  MoveL 658 to (4.03, 195.62, 30) mm, rotated rx 180 ry 50 rz -176.42 deg; joints [-18.981, -46.82, 111.254, 128.122, 73.547, 109.847, -1353.581]
  MoveL 659 to (9.5, 196.25, 40) mm, rotated rx 180 ry 50 rz -171.53 deg; joints [-18.576, -46.815, 111.235, 128.515, 73.401, 109.745, -1358.473]
  MoveL 660 to (15.19, 197.47, 50) mm, rotated rx -180 ry 50 rz -166.35 deg; joints [-18.172, -46.809, 111.211, 128.908, 73.253, 109.646, -1363.653]
  MoveL 661 to (21, 199.35, 60) mm, rotated rx -180 ry 50 rz -160.91 deg; joints [-17.768, -46.804, 111.18, 129.3, 73.102, 109.552, -1369.094]
  MoveL 662 to (26.8, 201.92, 70) mm, rotated rx 180 ry 50 rz -155.23 deg; joints [-17.364, -46.8, 111.144, 129.691, 72.947, 109.461, -1374.769]
  MoveL 663 to (32.46, 205.23, 80) mm, rotated rx -180 ry 50 rz -149.35 deg; joints [-16.96, -46.796, 111.102, 130.08, 72.788, 109.375, -1380.653]
  MoveL 664 to (37.86, 209.24, 90) mm, rotated rx 180 ry 50 rz -143.28 deg; joints [-16.557, -46.793, 111.054, 130.468, 72.625, 109.292, -1386.718]
  MoveL 665 to (42.85, 213.95, 100) mm, rotated rx 180 ry 50 rz -137.06 deg; joints [-16.154, -46.79, 110.999, 130.854, 72.459, 109.214, -1392.941]
  MoveL 666 to (47.33, 219.29, 110) mm, rotated rx -180 ry 50 rz -130.7 deg; joints [-15.751, -46.788, 110.939, 131.239, 72.288, 109.139, -1399.296]
  MoveL 667 to (51.17, 225.17, 120) mm, rotated rx -180 ry 50 rz -124.24 deg; joints [-15.349, -46.786, 110.873, 131.623, 72.114, 109.067, -1405.756]
  MoveL 668 to (54.3, 231.49, 130) mm, rotated rx -180 ry 50 rz -117.7 deg; joints [-14.948, -46.784, 110.801, 132.005, 71.937, 108.999, -1412.295]
  MoveL 669 to (56.65, 238.12, 140) mm, rotated rx 180 ry 50 rz -111.11 deg; joints [-14.546, -46.781, 110.723, 132.386, 71.756, 108.933, -1418.886]
  MoveL 670 to (58.18, 244.95, 150) mm, rotated rx 180 ry 50 rz -104.5 deg; joints [-14.146, -46.776, 110.639, 132.766, 71.573, 108.868, -1425.497]
  MoveL 671 to (58.89, 251.83, 160) mm, rotated rx 180 ry 50 rz -97.9 deg; joints [-13.746, -46.768, 110.548, 133.145, 71.387, 108.806, -1432.098]
  MoveL 672 to (58.8, 258.62, 170) mm, rotated rx -180 ry 50 rz -91.34 deg; joints [-13.346, -46.758, 110.451, 133.523, 71.199, 108.744, -1438.655]
  MoveL 673 to (57.96, 265.2, 180) mm, rotated rx 180 ry 50 rz -84.87 deg; joints [-12.947, -46.744, 110.348, 133.901, 71.009, 108.683, -1445.13]
  MoveL 674 to (56.44, 271.47, 190) mm, rotated rx 180 ry 50 rz -78.51 deg; joints [-12.549, -46.726, 110.239, 134.277, 70.818, 108.622, -1451.486]
  MoveL 675 to (54.33, 277.32, 200) mm, rotated rx -180 ry 50 rz -72.32 deg; joints [-12.152, -46.703, 110.123, 134.653, 70.627, 108.56, -1457.679]
  MoveL 676 to (51.74, 282.68, 210) mm, rotated rx 180 ry 50 rz -66.33 deg; joints [-11.755, -46.675, 110.001, 135.028, 70.435, 108.498, -1463.668]
  MoveL 677 to (48.8, 287.5, 220) mm, rotated rx -180 ry 50 rz -60.59 deg; joints [-11.359, -46.641, 109.872, 135.403, 70.242, 108.434, -1469.406]
  MoveL 678 to (45.62, 291.76, 230) mm, rotated rx 180 ry 50 rz -55.15 deg; joints [-10.964, -46.601, 109.737, 135.778, 70.049, 108.37, -1474.846]
  MoveL 679 to (42.34, 295.45, 240) mm, rotated rx 180 ry 50 rz -50.06 deg; joints [-10.57, -46.555, 109.596, 136.152, 69.856, 108.304, -1479.941]
  MoveL 680 to (39.07, 298.58, 250) mm, rotated rx 180 ry 50 rz -45.36 deg; joints [-10.177, -46.504, 109.448, 136.525, 69.663, 108.237, -1484.643]
  MoveL 681 to (35.92, 301.18, 260) mm, rotated rx -180 ry 50 rz -41.09 deg; joints [-9.784, -46.446, 109.294, 136.898, 69.47, 108.169, -1488.905]
  MoveL 682 to (33, 303.28, 270) mm, rotated rx 180 ry 50 rz -37.32 deg; joints [-9.393, -46.383, 109.133, 137.271, 69.277, 108.1, -1492.679]
  MoveL 683 to (30.4, 304.94, 280) mm, rotated rx 180 ry 50 rz -34.08 deg; joints [-9.003, -46.315, 108.966, 137.642, 69.083, 108.031, -1495.919]
  MoveL 684 to (28.22, 306.19, 290) mm, rotated rx 180 ry 50 rz -31.42 deg; joints [-8.613, -46.241, 108.793, 138.013, 68.889, 107.96, -1498.582]
  MoveL 685 to (-21.11, 309.47, 290) mm, rotated rx -180 ry 50 rz 23.11 deg; joints [-8.613, -46.26, 108.794, 138.009, 68.876, 107.972, -1553.11]
  Set speed (60.0 mm/s)
  MoveL 686 to (-18.74, 310.33, 280) mm, rotated rx -180 ry 50 rz 20.42 deg; joints [-9.003, -46.345, 108.968, 137.635, 69.063, 108.051, -1550.424]
  MoveL 687 to (-15.8, 311.23, 270) mm, rotated rx -180 ry 50 rz 17.14 deg; joints [-9.393, -46.428, 109.136, 137.26, 69.247, 108.13, -1547.138]
  MoveL 688 to (-12.3, 312.09, 260) mm, rotated rx 180 ry 50 rz 13.29 deg; joints [-9.784, -46.507, 109.298, 136.884, 69.429, 108.211, -1543.29]
  MoveL 689 to (-8.28, 312.8, 250) mm, rotated rx -180 ry 50 rz 8.92 deg; joints [-10.177, -46.583, 109.454, 136.506, 69.61, 108.292, -1538.917]
  MoveL 690 to (-3.78, 313.26, 240) mm, rotated rx -180 ry 50 rz 4.06 deg; joints [-10.57, -46.655, 109.603, 136.128, 69.79, 108.372, -1534.059]
  MoveL 691 to (1.16, 313.37, 230) mm, rotated rx 180 ry 50 rz -1.24 deg; joints [-10.964, -46.722, 109.746, 135.749, 69.969, 108.453, -1528.756]
  MoveL 692 to (6.46, 313.03, 220) mm, rotated rx 180 ry 50 rz -6.95 deg; joints [-11.359, -46.783, 109.883, 135.37, 70.148, 108.533, -1523.053]
  MoveL 693 to (12.04, 312.14, 210) mm, rotated rx 180 ry 50 rz -13.01 deg; joints [-11.755, -46.838, 110.013, 134.99, 70.327, 108.612, -1516.995]
  MoveL 694 to (17.8, 310.63, 200) mm, rotated rx 180 ry 50 rz -19.37 deg; joints [-12.152, -46.887, 110.136, 134.61, 70.507, 108.689, -1510.629]
  MoveL 695 to (23.62, 308.44, 190) mm, rotated rx -180 ry 50 rz -25.99 deg; joints [-12.549, -46.929, 110.254, 134.23, 70.687, 108.765, -1504.006]
  MoveL 696 to (29.38, 305.54, 180) mm, rotated rx -180 ry 50 rz -32.82 deg; joints [-12.947, -46.964, 110.364, 133.85, 70.868, 108.838, -1497.176]
  MoveL 697 to (34.94, 301.92, 170) mm, rotated rx -180 ry 50 rz -39.81 deg; joints [-13.346, -46.992, 110.469, 133.47, 71.049, 108.911, -1490.188]
  MoveL 698 to (40.17, 297.58, 160) mm, rotated rx 180 ry 50 rz -46.91 deg; joints [-13.746, -47.014, 110.566, 133.089, 71.231, 108.981, -1483.094]
  MoveL 699 to (44.94, 292.58, 150) mm, rotated rx -180 ry 50 rz -54.06 deg; joints [-14.146, -47.029, 110.658, 132.709, 71.413, 109.05, -1475.941]
  MoveL 700 to (49.15, 286.99, 140) mm, rotated rx -180 ry 50 rz -61.23 deg; joints [-14.546, -47.038, 110.743, 132.328, 71.596, 109.118, -1468.774]
  MoveL 701 to (52.68, 280.9, 130) mm, rotated rx -180 ry 50 rz -68.36 deg; joints [-14.948, -47.042, 110.821, 131.947, 71.777, 109.185, -1461.638]
  MoveL 702 to (55.46, 274.42, 120) mm, rotated rx -180 ry 50 rz -75.43 deg; joints [-15.349, -47.042, 110.893, 131.566, 71.958, 109.252, -1454.572]
  MoveL 703 to (57.44, 267.68, 110) mm, rotated rx 180 ry 50 rz -82.39 deg; joints [-15.751, -47.037, 110.959, 131.184, 72.137, 109.32, -1447.613]
  MoveL 704 to (58.6, 260.81, 100) mm, rotated rx 180 ry 50 rz -89.21 deg; joints [-16.154, -47.029, 111.018, 130.801, 72.315, 109.388, -1440.794]
  MoveL 705 to (58.95, 253.96, 90) mm, rotated rx -180 ry 50 rz -95.85 deg; joints [-16.557, -47.019, 111.072, 130.418, 72.49, 109.458, -1434.147]
  MoveL 706 to (58.51, 247.24, 80) mm, rotated rx -180 ry 50 rz -102.3 deg; joints [-16.96, -47.007, 111.119, 130.034, 72.663, 109.53, -1427.701]
  MoveL 707 to (57.35, 240.79, 70) mm, rotated rx 180 ry 50 rz -108.52 deg; joints [-17.364, -46.993, 111.16, 129.648, 72.833, 109.604, -1421.482]
  MoveL 708 to (55.55, 234.7, 60) mm, rotated rx -180 ry 50 rz -114.48 deg; joints [-17.768, -46.979, 111.195, 129.262, 73, 109.682, -1415.517]
  MoveL 709 to (53.21, 229.07, 50) mm, rotated rx 180 ry 50 rz -120.17 deg; joints [-18.172, -46.965, 111.224, 128.875, 73.164, 109.762, -1409.83]
  MoveL 710 to (50.45, 223.94, 40) mm, rotated rx 180 ry 50 rz -125.55 deg; joints [-18.576, -46.951, 111.246, 128.486, 73.324, 109.847, -1404.447]
  MoveL 711 to (47.39, 219.37, 30) mm, rotated rx 180 ry 50 rz -130.61 deg; joints [-18.981, -46.936, 111.263, 128.097, 73.481, 109.934, -1399.391]
  MoveL 712 to (44.15, 215.37, 20) mm, rotated rx 180 ry 50 rz -135.31 deg; joints [-19.385, -46.922, 111.274, 127.706, 73.634, 110.026, -1394.688]
  MoveL 713 to (40.85, 211.93, 10) mm, rotated rx 180 ry 50 rz -139.64 deg; joints [-19.79, -46.908, 111.279, 127.315, 73.785, 110.121, -1390.363]
  MoveL 714 to (37.62, 209.05, 0) mm, rotated rx 180 ry 50 rz -143.56 deg; joints [-20.194, -46.894, 111.278, 126.922, 73.932, 110.22, -1386.442]
  MoveL 715 to (-21.11, 309.47, 290) mm, rotated rx -180 ry 50 rz 23.11 deg; joints [-8.613, -46.26, 108.794, 138.009, 68.876, 107.972, -1553.11]
  Set speed (60.0 mm/s)
  MoveL 716 to (-34.79, 325.15, 290) mm, rotated rx 180 ry 50 rz 28.1 deg; joints [-8.613, -45.167, 108.701, 138.262, 69.621, 107.259, -1558.101]
  MoveL 717 to (37.62, 209.05, 0) mm, rotated rx 180 ry 50 rz -143.56 deg; joints [-20.194, -46.894, 111.278, 126.922, 73.932, 110.22, -1386.442]
  Set speed (60.0 mm/s)
  MoveL 718 to (55.59, 198.58, 0) mm, rotated rx 180 ry 50 rz -137.85 deg; joints [-20.194, -45.798, 111.172, 127.145, 74.528, 109.399, -1392.15]
  MoveL 719 to (37.62, 209.05, 0) mm, rotated rx 180 ry 50 rz -143.56 deg; joints [-20.194, -46.894, 111.278, 126.922, 73.932, 110.22, -1386.442]
  Set speed (60.0 mm/s)
  MoveL 720 to (40.85, 211.93, 10) mm, rotated rx 180 ry 50 rz -139.64 deg; joints [-19.79, -46.908, 111.279, 127.315, 73.785, 110.121, -1390.363]
  MoveL 721 to (44.15, 215.37, 20) mm, rotated rx 180 ry 50 rz -135.31 deg; joints [-19.385, -46.922, 111.274, 127.706, 73.634, 110.026, -1394.688]
  MoveL 722 to (47.39, 219.37, 30) mm, rotated rx 180 ry 50 rz -130.61 deg; joints [-18.981, -46.936, 111.263, 128.097, 73.481, 109.934, -1399.391]
  MoveL 723 to (50.45, 223.94, 40) mm, rotated rx 180 ry 50 rz -125.55 deg; joints [-18.576, -46.951, 111.246, 128.486, 73.324, 109.847, -1404.447]
  MoveL 724 to (53.21, 229.07, 50) mm, rotated rx 180 ry 50 rz -120.17 deg; joints [-18.172, -46.965, 111.224, 128.875, 73.164, 109.762, -1409.83]
  MoveL 725 to (55.55, 234.7, 60) mm, rotated rx -180 ry 50 rz -114.48 deg; joints [-17.768, -46.979, 111.195, 129.262, 73, 109.682, -1415.517]
  MoveL 726 to (57.35, 240.79, 70) mm, rotated rx -180 ry 50 rz -108.52 deg; joints [-17.364, -46.993, 111.16, 129.648, 72.833, 109.604, -1421.482]
  MoveL 727 to (58.51, 247.24, 80) mm, rotated rx 180 ry 50 rz -102.3 deg; joints [-16.96, -47.007, 111.119, 130.034, 72.663, 109.53, -1427.701]
  MoveL 728 to (58.95, 253.96, 90) mm, rotated rx 180 ry 50 rz -95.85 deg; joints [-16.557, -47.019, 111.072, 130.418, 72.49, 109.458, -1434.147]
  MoveL 729 to (58.6, 260.81, 100) mm, rotated rx 180 ry 50 rz -89.21 deg; joints [-16.154, -47.029, 111.018, 130.801, 72.315, 109.388, -1440.794]
  MoveL 730 to (57.44, 267.68, 110) mm, rotated rx 180 ry 50 rz -82.39 deg; joints [-15.751, -47.037, 110.959, 131.184, 72.137, 109.32, -1447.613]
  MoveL 731 to (55.46, 274.42, 120) mm, rotated rx 180 ry 50 rz -75.43 deg; joints [-15.349, -47.042, 110.893, 131.566, 71.958, 109.252, -1454.572]
  MoveL 732 to (52.68, 280.9, 130) mm, rotated rx -180 ry 50 rz -68.36 deg; joints [-14.948, -47.042, 110.821, 131.947, 71.777, 109.185, -1461.638]
  MoveL 733 to (49.15, 286.99, 140) mm, rotated rx -180 ry 50 rz -61.23 deg; joints [-14.546, -47.038, 110.743, 132.328, 71.596, 109.118, -1468.774]
  MoveL 734 to (44.94, 292.58, 150) mm, rotated rx -180 ry 50 rz -54.06 deg; joints [-14.146, -47.029, 110.658, 132.709, 71.413, 109.05, -1475.941]
  MoveL 735 to (40.17, 297.58, 160) mm, rotated rx -180 ry 50 rz -46.91 deg; joints [-13.746, -47.014, 110.566, 133.089, 71.231, 108.981, -1483.094]
  MoveL 736 to (34.94, 301.92, 170) mm, rotated rx 180 ry 50 rz -39.81 deg; joints [-13.346, -46.992, 110.469, 133.47, 71.049, 108.911, -1490.188]
  MoveL 737 to (29.38, 305.54, 180) mm, rotated rx 180 ry 50 rz -32.82 deg; joints [-12.947, -46.964, 110.364, 133.85, 70.868, 108.838, -1497.176]
  MoveL 738 to (23.62, 308.44, 190) mm, rotated rx 180 ry 50 rz -25.99 deg; joints [-12.549, -46.929, 110.254, 134.23, 70.687, 108.765, -1504.006]
  MoveL 739 to (17.8, 310.63, 200) mm, rotated rx -180 ry 50 rz -19.37 deg; joints [-12.152, -46.887, 110.136, 134.61, 70.507, 108.689, -1510.629]
  MoveL 740 to (12.04, 312.14, 210) mm, rotated rx 180 ry 50 rz -13.01 deg; joints [-11.755, -46.838, 110.013, 134.99, 70.327, 108.612, -1516.995]
  MoveL 741 to (6.46, 313.03, 220) mm, rotated rx 180 ry 50 rz -6.95 deg; joints [-11.359, -46.783, 109.883, 135.37, 70.148, 108.533, -1523.053]
  MoveL 742 to (1.16, 313.37, 230) mm, rotated rx 180 ry 50 rz -1.24 deg; joints [-10.964, -46.722, 109.746, 135.749, 69.969, 108.453, -1528.756]
  MoveL 743 to (-3.78, 313.26, 240) mm, rotated rx 180 ry 50 rz 4.06 deg; joints [-10.57, -46.655, 109.603, 136.128, 69.79, 108.372, -1534.059]
  MoveL 744 to (-8.28, 312.8, 250) mm, rotated rx 180 ry 50 rz 8.92 deg; joints [-10.177, -46.583, 109.454, 136.506, 69.61, 108.292, -1538.917]
  MoveL 745 to (-12.3, 312.09, 260) mm, rotated rx -180 ry 50 rz 13.29 deg; joints [-9.784, -46.507, 109.298, 136.884, 69.429, 108.211, -1543.29]
  MoveL 746 to (-15.8, 311.23, 270) mm, rotated rx -180 ry 50 rz 17.14 deg; joints [-9.393, -46.428, 109.136, 137.26, 69.247, 108.13, -1547.138]
  MoveL 747 to (-18.74, 310.33, 280) mm, rotated rx -180 ry 50 rz 20.42 deg; joints [-9.003, -46.345, 108.968, 137.635, 69.063, 108.051, -1550.424]
  MoveL 748 to (-21.11, 309.47, 290) mm, rotated rx -180 ry 50 rz 23.11 deg; joints [-8.613, -46.26, 108.794, 138.009, 68.876, 107.972, -1553.11]
  MoveL 749 to (-34.79, 325.15, 290) mm, rotated rx 180 ry 50 rz 28.1 deg; joints [-8.613, -45.167, 108.701, 138.262, 69.621, 107.259, -1558.101]
  Set speed (60.0 mm/s)
  MoveL 750 to (-31.73, 326.57, 280) mm, rotated rx 180 ry 50 rz 25.49 deg; joints [-9.003, -45.252, 108.876, 137.888, 69.803, 107.332, -1555.486]
  MoveL 751 to (-27.92, 328.13, 270) mm, rotated rx -180 ry 50 rz 22.29 deg; joints [-9.393, -45.334, 109.044, 137.512, 69.984, 107.407, -1552.288]
  MoveL 752 to (-23.38, 329.69, 260) mm, rotated rx 180 ry 50 rz 18.54 deg; joints [-9.784, -45.413, 109.206, 137.135, 70.162, 107.483, -1548.542]
  MoveL 753 to (-18.11, 331.13, 250) mm, rotated rx 180 ry 50 rz 14.29 deg; joints [-10.177, -45.49, 109.362, 136.757, 70.338, 107.56, -1544.286]
  MoveL 754 to (-12.17, 332.29, 240) mm, rotated rx -180 ry 50 rz 9.56 deg; joints [-10.57, -45.562, 109.511, 136.378, 70.513, 107.636, -1539.557]
  MoveL 755 to (-5.61, 333.04, 230) mm, rotated rx -180 ry 50 rz 4.39 deg; joints [-10.964, -45.629, 109.655, 135.998, 70.687, 107.713, -1534.392]
  MoveL 756 to (1.49, 333.22, 220) mm, rotated rx 180 ry 50 rz -1.17 deg; joints [-11.359, -45.692, 109.791, 135.618, 70.861, 107.79, -1528.834]
  MoveL 757 to (9.03, 332.72, 210) mm, rotated rx 180 ry 50 rz -7.08 deg; joints [-11.755, -45.749, 109.922, 135.237, 71.034, 107.865, -1522.922]
  MoveL 758 to (16.88, 331.41, 200) mm, rotated rx -180 ry 50 rz -13.3 deg; joints [-12.152, -45.799, 110.045, 134.856, 71.208, 107.94, -1516.702]
  MoveL 759 to (24.89, 329.2, 190) mm, rotated rx -180 ry 50 rz -19.78 deg; joints [-12.549, -45.843, 110.162, 134.474, 71.382, 108.013, -1510.217]
  MoveL 760 to (32.91, 326.04, 180) mm, rotated rx 180 ry 50 rz -26.49 deg; joints [-12.947, -45.88, 110.273, 134.093, 71.557, 108.084, -1503.513]
  MoveL 761 to (40.75, 321.89, 170) mm, rotated rx 180 ry 50 rz -33.36 deg; joints [-13.346, -45.91, 110.377, 133.711, 71.732, 108.154, -1496.637]
  MoveL 762 to (48.24, 316.75, 160) mm, rotated rx -180 ry 50 rz -40.37 deg; joints [-13.746, -45.934, 110.474, 133.329, 71.908, 108.222, -1489.635]
  MoveL 763 to (55.2, 310.67, 150) mm, rotated rx -180 ry 50 rz -47.45 deg; joints [-14.146, -45.95, 110.565, 132.947, 72.084, 108.289, -1482.551]
  MoveL 764 to (61.48, 303.74, 140) mm, rotated rx -180 ry 50 rz -54.57 deg; joints [-14.546, -45.961, 110.649, 132.565, 72.26, 108.354, -1475.431]
  MoveL 765 to (66.92, 296.06, 130) mm, rotated rx -180 ry 50 rz -61.68 deg; joints [-14.948, -45.965, 110.727, 132.183, 72.436, 108.419, -1468.317]
  MoveL 766 to (71.41, 287.77, 120) mm, rotated rx 180 ry 50 rz -68.75 deg; joints [-15.349, -45.965, 110.798, 131.8, 72.611, 108.483, -1461.249]
  MoveL 767 to (74.87, 279.04, 110) mm, rotated rx -180 ry 50 rz -75.73 deg; joints [-15.751, -45.96, 110.863, 131.417, 72.785, 108.547, -1454.266]
  MoveL 768 to (77.24, 270.04, 100) mm, rotated rx 180 ry 50 rz -82.6 deg; joints [-16.154, -45.952, 110.921, 131.033, 72.957, 108.612, -1447.404]
  MoveL 769 to (78.53, 260.95, 90) mm, rotated rx -180 ry 50 rz -89.3 deg; joints [-16.557, -45.941, 110.974, 130.648, 73.127, 108.678, -1440.696]
  MoveL 770 to (78.77, 251.96, 80) mm, rotated rx 180 ry 50 rz -95.83 deg; joints [-16.96, -45.927, 111.02, 130.263, 73.295, 108.746, -1434.174]
  MoveL 771 to (78, 243.23, 70) mm, rotated rx -180 ry 50 rz -102.13 deg; joints [-17.364, -45.912, 111.06, 129.877, 73.461, 108.816, -1427.868]
  MoveL 772 to (76.35, 234.91, 60) mm, rotated rx -180 ry 50 rz -108.19 deg; joints [-17.768, -45.896, 111.093, 129.49, 73.623, 108.889, -1421.808]
  MoveL 773 to (73.92, 227.12, 50) mm, rotated rx 180 ry 50 rz -113.98 deg; joints [-18.172, -45.88, 111.121, 129.101, 73.782, 108.965, -1416.021]
  MoveL 774 to (70.87, 219.96, 40) mm, rotated rx -180 ry 50 rz -119.46 deg; joints [-18.576, -45.863, 111.143, 128.712, 73.938, 109.045, -1410.535]
  MoveL 775 to (67.34, 213.5, 30) mm, rotated rx 180 ry 50 rz -124.62 deg; joints [-18.981, -45.847, 111.159, 128.322, 74.09, 109.128, -1405.378]
  MoveL 776 to (63.51, 207.78, 20) mm, rotated rx 180 ry 50 rz -129.42 deg; joints [-19.385, -45.83, 111.17, 127.931, 74.24, 109.214, -1400.576]
  MoveL 777 to (59.54, 202.81, 10) mm, rotated rx 180 ry 50 rz -133.84 deg; joints [-19.79, -45.814, 111.174, 127.539, 74.386, 109.305, -1396.157]
  MoveL 778 to (55.59, 198.58, 0) mm, rotated rx -180 ry 50 rz -137.85 deg; joints [-20.194, -45.798, 111.172, 127.145, 74.528, 109.399, -1392.15]
  MoveL 779 to (-34.79, 325.15, 290) mm, rotated rx 180 ry 50 rz 28.1 deg; joints [-8.613, -45.167, 108.701, 138.262, 69.621, 107.259, -1558.101]
  Set speed (60.0 mm/s)
  MoveL 780 to (-30.72, 304.75, 290) mm, rotated rx 180 ry 50 rz 34.47 deg; joints [-8.613, -46.233, 108.792, 138.015, 68.894, 107.955, -1564.467]
  MoveL 781 to (55.59, 198.58, 0) mm, rotated rx 180 ry 50 rz -137.85 deg; joints [-20.194, -45.798, 111.172, 127.145, 74.528, 109.399, -1392.15]
  Set speed (60.0 mm/s)
  MoveL 782 to (45.21, 216.6, 0) mm, rotated rx -180 ry 50 rz -133.83 deg; joints [-20.194, -46.931, 111.281, 126.914, 73.912, 110.249, -1396.169]
  MoveL 783 to (55.59, 198.58, 0) mm, rotated rx -180 ry 50 rz -137.85 deg; joints [-20.194, -45.798, 111.172, 127.145, 74.528, 109.399, -1392.15]
  Set speed (60.0 mm/s)
  MoveL 784 to (59.54, 202.81, 10) mm, rotated rx 180 ry 50 rz -133.84 deg; joints [-19.79, -45.814, 111.174, 127.539, 74.386, 109.305, -1396.157]
  MoveL 785 to (63.51, 207.78, 20) mm, rotated rx -180 ry 50 rz -129.42 deg; joints [-19.385, -45.83, 111.17, 127.931, 74.24, 109.214, -1400.576]
  MoveL 786 to (67.34, 213.5, 30) mm, rotated rx 180 ry 50 rz -124.62 deg; joints [-18.981, -45.847, 111.159, 128.322, 74.09, 109.128, -1405.378]
  MoveL 787 to (70.87, 219.96, 40) mm, rotated rx -180 ry 50 rz -119.46 deg; joints [-18.576, -45.863, 111.143, 128.712, 73.938, 109.045, -1410.535]
  MoveL 788 to (73.92, 227.12, 50) mm, rotated rx -180 ry 50 rz -113.98 deg; joints [-18.172, -45.88, 111.121, 129.101, 73.782, 108.965, -1416.021]
  MoveL 789 to (76.35, 234.91, 60) mm, rotated rx 180 ry 50 rz -108.19 deg; joints [-17.768, -45.896, 111.093, 129.49, 73.623, 108.889, -1421.808]
  MoveL 790 to (78, 243.23, 70) mm, rotated rx 180 ry 50 rz -102.13 deg; joints [-17.364, -45.912, 111.06, 129.877, 73.461, 108.816, -1427.868]
  MoveL 791 to (78.77, 251.96, 80) mm, rotated rx -180 ry 50 rz -95.83 deg; joints [-16.96, -45.927, 111.02, 130.263, 73.295, 108.746, -1434.174]
  MoveL 792 to (78.53, 260.95, 90) mm, rotated rx 180 ry 50 rz -89.3 deg; joints [-16.557, -45.941, 110.974, 130.648, 73.127, 108.678, -1440.696]
  MoveL 793 to (77.24, 270.04, 100) mm, rotated rx -180 ry 50 rz -82.6 deg; joints [-16.154, -45.952, 110.921, 131.033, 72.957, 108.612, -1447.404]
  MoveL 794 to (74.87, 279.04, 110) mm, rotated rx -180 ry 50 rz -75.73 deg; joints [-15.751, -45.96, 110.863, 131.417, 72.785, 108.547, -1454.266]
  MoveL 795 to (71.41, 287.77, 120) mm, rotated rx -180 ry 50 rz -68.75 deg; joints [-15.349, -45.965, 110.798, 131.8, 72.611, 108.483, -1461.249]
  MoveL 796 to (66.92, 296.06, 130) mm, rotated rx -180 ry 50 rz -61.68 deg; joints [-14.948, -45.965, 110.727, 132.183, 72.436, 108.419, -1468.317]
  MoveL 797 to (61.48, 303.74, 140) mm, rotated rx -180 ry 50 rz -54.57 deg; joints [-14.546, -45.961, 110.649, 132.565, 72.26, 108.354, -1475.431]
  MoveL 798 to (55.2, 310.67, 150) mm, rotated rx 180 ry 50 rz -47.45 deg; joints [-14.146, -45.95, 110.565, 132.947, 72.084, 108.289, -1482.551]
  MoveL 799 to (48.24, 316.75, 160) mm, rotated rx -180 ry 50 rz -40.37 deg; joints [-13.746, -45.934, 110.474, 133.329, 71.908, 108.222, -1489.635]
  MoveL 800 to (40.75, 321.89, 170) mm, rotated rx -180 ry 50 rz -33.36 deg; joints [-13.346, -45.91, 110.377, 133.711, 71.732, 108.154, -1496.637]
  MoveL 801 to (32.91, 326.04, 180) mm, rotated rx -180 ry 50 rz -26.49 deg; joints [-12.947, -45.88, 110.273, 134.093, 71.557, 108.084, -1503.513]
  MoveL 802 to (24.89, 329.2, 190) mm, rotated rx 180 ry 50 rz -19.78 deg; joints [-12.549, -45.843, 110.162, 134.474, 71.382, 108.013, -1510.217]
  MoveL 803 to (16.88, 331.41, 200) mm, rotated rx -180 ry 50 rz -13.3 deg; joints [-12.152, -45.799, 110.045, 134.856, 71.208, 107.94, -1516.702]
  MoveL 804 to (9.03, 332.72, 210) mm, rotated rx -180 ry 50 rz -7.08 deg; joints [-11.755, -45.749, 109.922, 135.237, 71.034, 107.865, -1522.922]
  MoveL 805 to (1.49, 333.22, 220) mm, rotated rx -180 ry 50 rz -1.17 deg; joints [-11.359, -45.692, 109.791, 135.618, 70.861, 107.79, -1528.834]
  MoveL 806 to (-5.61, 333.04, 230) mm, rotated rx 180 ry 50 rz 4.39 deg; joints [-10.964, -45.629, 109.655, 135.998, 70.687, 107.713, -1534.392]
  MoveL 807 to (-12.17, 332.29, 240) mm, rotated rx -180 ry 50 rz 9.56 deg; joints [-10.57, -45.562, 109.511, 136.378, 70.513, 107.636, -1539.557]
  MoveL 808 to (-18.11, 331.13, 250) mm, rotated rx -180 ry 50 rz 14.29 deg; joints [-10.177, -45.49, 109.362, 136.757, 70.338, 107.56, -1544.286]
  MoveL 809 to (-23.38, 329.69, 260) mm, rotated rx 180 ry 50 rz 18.54 deg; joints [-9.784, -45.413, 109.206, 137.135, 70.162, 107.483, -1548.542]
  MoveL 810 to (-27.92, 328.13, 270) mm, rotated rx -180 ry 50 rz 22.29 deg; joints [-9.393, -45.334, 109.044, 137.512, 69.984, 107.407, -1552.288]
  MoveL 811 to (-31.73, 326.57, 280) mm, rotated rx -180 ry 50 rz 25.49 deg; joints [-9.003, -45.252, 108.876, 137.888, 69.803, 107.332, -1555.486]
  MoveL 812 to (-34.79, 325.15, 290) mm, rotated rx 180 ry 50 rz 28.1 deg; joints [-8.613, -45.167, 108.701, 138.262, 69.621, 107.259, -1558.101]
  MoveL 813 to (-30.72, 304.75, 290) mm, rotated rx 180 ry 50 rz 34.47 deg; joints [-8.613, -46.233, 108.792, 138.015, 68.894, 107.955, -1564.467]
  Set speed (60.0 mm/s)
  MoveL 814 to (-28.54, 306.02, 280) mm, rotated rx -180 ry 50 rz 31.81 deg; joints [-9.003, -46.321, 108.967, 137.641, 69.079, 108.035, -1561.806]
  MoveL 815 to (-25.81, 307.44, 270) mm, rotated rx -180 ry 50 rz 28.55 deg; joints [-9.393, -46.406, 109.135, 137.265, 69.261, 108.116, -1558.548]
  MoveL 816 to (-22.53, 308.91, 260) mm, rotated rx -180 ry 50 rz 24.73 deg; joints [-9.784, -46.489, 109.297, 136.888, 69.441, 108.199, -1554.728]
  MoveL 817 to (-18.7, 310.34, 250) mm, rotated rx 180 ry 50 rz 20.38 deg; joints [-10.177, -46.569, 109.453, 136.51, 69.619, 108.282, -1550.381]
  MoveL 818 to (-14.35, 311.61, 240) mm, rotated rx 180 ry 50 rz 15.54 deg; joints [-10.57, -46.645, 109.602, 136.131, 69.796, 108.366, -1545.543]
  MoveL 819 to (-9.52, 312.61, 230) mm, rotated rx 180 ry 50 rz 10.25 deg; joints [-10.964, -46.717, 109.746, 135.75, 69.972, 108.45, -1540.254]
  MoveL 820 to (-4.24, 313.23, 220) mm, rotated rx -180 ry 50 rz 4.55 deg; joints [-11.359, -46.784, 109.883, 135.37, 70.147, 108.534, -1534.554]
  MoveL 821 to (1.41, 313.37, 210) mm, rotated rx 180 ry 50 rz -1.51 deg; joints [-11.755, -46.845, 110.013, 134.989, 70.323, 108.616, -1528.487]
  MoveL 822 to (7.35, 312.92, 200) mm, rotated rx 180 ry 50 rz -7.9 deg; joints [-12.152, -46.9, 110.137, 134.607, 70.498, 108.698, -1522.098]
  MoveL 823 to (13.47, 311.83, 190) mm, rotated rx 180 ry 50 rz -14.57 deg; joints [-12.549, -46.948, 110.255, 134.226, 70.675, 108.778, -1515.435]
  MoveL 824 to (19.65, 310.01, 180) mm, rotated rx 180 ry 50 rz -21.45 deg; joints [-12.947, -46.989, 110.366, 133.844, 70.852, 108.856, -1508.548]
  MoveL 825 to (25.78, 307.45, 170) mm, rotated rx 180 ry 50 rz -28.51 deg; joints [-13.346, -47.024, 110.471, 133.462, 71.029, 108.933, -1501.489]
  MoveL 826 to (31.7, 304.13, 160) mm, rotated rx -180 ry 50 rz -35.69 deg; joints [-13.746, -47.051, 110.569, 133.081, 71.208, 109.007, -1494.307]
  MoveL 827 to (37.3, 300.08, 150) mm, rotated rx 180 ry 50 rz -42.95 deg; joints [-14.146, -47.071, 110.661, 132.699, 71.387, 109.08, -1487.054]
  MoveL 828 to (42.45, 295.34, 140) mm, rotated rx 180 ry 50 rz -50.22 deg; joints [-14.546, -47.085, 110.746, 132.318, 71.567, 109.151, -1479.778]
  MoveL 829 to (47.02, 289.99, 130) mm, rotated rx 180 ry 50 rz -57.48 deg; joints [-14.948, -47.092, 110.825, 131.936, 71.746, 109.221, -1472.524]
  MoveL 830 to (50.93, 284.12, 120) mm, rotated rx -180 ry 50 rz -64.66 deg; joints [-15.349, -47.094, 110.897, 131.554, 71.926, 109.291, -1465.337]
  MoveL 831 to (54.1, 277.85, 110) mm, rotated rx -180 ry 50 rz -71.74 deg; joints [-15.751, -47.092, 110.963, 131.172, 72.104, 109.36, -1458.256]
  MoveL 832 to (56.49, 271.3, 100) mm, rotated rx 180 ry 50 rz -78.68 deg; joints [-16.154, -47.085, 111.023, 130.789, 72.281, 109.429, -1451.316]
  MoveL 833 to (58.06, 264.62, 90) mm, rotated rx 180 ry 50 rz -85.45 deg; joints [-16.557, -47.075, 111.076, 130.405, 72.457, 109.499, -1444.553]
  MoveL 834 to (58.85, 257.94, 80) mm, rotated rx -180 ry 50 rz -92 deg; joints [-16.96, -47.062, 111.123, 130.021, 72.63, 109.571, -1437.997]
  MoveL 835 to (58.87, 251.39, 70) mm, rotated rx 180 ry 50 rz -98.32 deg; joints [-17.364, -47.048, 111.164, 129.636, 72.801, 109.645, -1431.675]
  MoveL 836 to (58.2, 245.07, 60) mm, rotated rx 180 ry 50 rz -104.38 deg; joints [-17.768, -47.032, 111.199, 129.251, 72.969, 109.721, -1425.616]
  MoveL 837 to (56.92, 239.11, 50) mm, rotated rx 180 ry 50 rz -110.16 deg; joints [-18.172, -47.016, 111.228, 128.864, 73.134, 109.801, -1419.845]
  MoveL 838 to (55.13, 233.57, 40) mm, rotated rx -180 ry 50 rz -115.61 deg; joints [-18.576, -46.999, 111.25, 128.476, 73.296, 109.883, -1414.385]
  MoveL 839 to (52.95, 228.52, 30) mm, rotated rx -180 ry 50 rz -120.74 deg; joints [-18.981, -46.982, 111.267, 128.087, 73.455, 109.969, -1409.263]
  MoveL 840 to (50.48, 223.99, 20) mm, rotated rx 180 ry 50 rz -125.5 deg; joints [-19.385, -46.965, 111.278, 127.697, 73.61, 110.058, -1404.503]
  MoveL 841 to (47.86, 220.02, 10) mm, rotated rx 180 ry 50 rz -129.87 deg; joints [-19.79, -46.948, 111.283, 127.306, 73.762, 110.152, -1400.13]
  MoveL 842 to (45.21, 216.6, 0) mm, rotated rx 180 ry 50 rz -133.83 deg; joints [-20.194, -46.931, 111.281, 126.914, 73.912, 110.249, -1396.169]
  MoveL 843 to (-30.72, 304.75, 290) mm, rotated rx -180 ry 50 rz 34.47 deg; joints [-8.613, -46.233, 108.792, 138.015, 68.894, 107.955, -1564.467]
  Set speed (60.0 mm/s)
  MoveL 844 to (-58.22, 263.67, 290) mm, rotated rx -180 ry 50 rz 86.39 deg; joints [-8.613, -46.013, 108.776, 138.068, 69.046, 107.809, -1616.394]
  MoveL 845 to (45.21, 216.6, 0) mm, rotated rx 180 ry 50 rz -133.83 deg; joints [-20.194, -46.931, 111.281, 126.914, 73.912, 110.249, -1756.169]
  Set speed (60.0 mm/s)
  MoveL 846 to (58.12, 264.32, 0) mm, rotated rx -180 ry 50 rz -85.75 deg; joints [-20.194, -47.176, 111.301, 126.862, 73.776, 110.437, -1804.254]
  MoveL 847 to (45.21, 216.6, 0) mm, rotated rx -180 ry 50 rz -133.83 deg; joints [-20.194, -46.931, 111.281, 126.914, 73.912, 110.249, -1756.169]
  Set speed (60.0 mm/s)
  MoveL 848 to (47.86, 220.02, 10) mm, rotated rx -180 ry 50 rz -129.87 deg; joints [-19.79, -46.948, 111.283, 127.306, 73.762, 110.152, -1760.13]
  MoveL 849 to (50.48, 223.99, 20) mm, rotated rx 180 ry 50 rz -125.5 deg; joints [-19.385, -46.965, 111.278, 127.697, 73.61, 110.058, -1764.503]
  MoveL 850 to (52.95, 228.52, 30) mm, rotated rx 180 ry 50 rz -120.74 deg; joints [-18.981, -46.982, 111.267, 128.087, 73.455, 109.969, -1769.263]
  MoveL 851 to (55.13, 233.57, 40) mm, rotated rx -180 ry 50 rz -115.61 deg; joints [-18.576, -46.999, 111.25, 128.476, 73.296, 109.883, -1774.385]
  MoveL 852 to (56.92, 239.11, 50) mm, rotated rx 180 ry 50 rz -110.16 deg; joints [-18.172, -47.016, 111.228, 128.864, 73.134, 109.801, -1779.845]
  MoveL 853 to (58.2, 245.07, 60) mm, rotated rx 180 ry 50 rz -104.38 deg; joints [-17.768, -47.032, 111.199, 129.251, 72.969, 109.721, -1785.616]
  MoveL 854 to (58.87, 251.39, 70) mm, rotated rx 180 ry 50 rz -98.32 deg; joints [-17.364, -47.048, 111.164, 129.636, 72.801, 109.645, -1791.675]
  MoveL 855 to (58.85, 257.94, 80) mm, rotated rx -180 ry 50 rz -92 deg; joints [-16.96, -47.062, 111.123, 130.021, 72.63, 109.571, -1797.997]
  MoveL 856 to (58.06, 264.62, 90) mm, rotated rx 180 ry 50 rz -85.45 deg; joints [-16.557, -47.075, 111.076, 130.405, 72.457, 109.499, -1804.553]
  MoveL 857 to (56.49, 271.3, 100) mm, rotated rx 180 ry 50 rz -78.68 deg; joints [-16.154, -47.085, 111.023, 130.789, 72.281, 109.429, -1811.316]
  MoveL 858 to (54.1, 277.85, 110) mm, rotated rx -180 ry 50 rz -71.74 deg; joints [-15.751, -47.092, 110.963, 131.172, 72.104, 109.36, -1818.256]
  MoveL 859 to (50.93, 284.12, 120) mm, rotated rx -180 ry 50 rz -64.66 deg; joints [-15.349, -47.094, 110.897, 131.554, 71.926, 109.291, -1825.337]
  MoveL 860 to (47.02, 289.99, 130) mm, rotated rx -180 ry 50 rz -57.48 deg; joints [-14.948, -47.092, 110.825, 131.936, 71.746, 109.221, -1832.524]
  MoveL 861 to (42.45, 295.34, 140) mm, rotated rx 180 ry 50 rz -50.22 deg; joints [-14.546, -47.085, 110.746, 132.318, 71.567, 109.151, -1839.778]
  MoveL 862 to (37.3, 300.08, 150) mm, rotated rx -180 ry 50 rz -42.95 deg; joints [-14.146, -47.071, 110.661, 132.699, 71.387, 109.08, -1847.054]
  MoveL 863 to (31.7, 304.13, 160) mm, rotated rx -180 ry 50 rz -35.69 deg; joints [-13.746, -47.051, 110.569, 133.081, 71.208, 109.007, -1854.307]
  MoveL 864 to (25.78, 307.45, 170) mm, rotated rx -180 ry 50 rz -28.51 deg; joints [-13.346, -47.024, 110.471, 133.462, 71.029, 108.933, -1861.489]
  MoveL 865 to (19.65, 310.01, 180) mm, rotated rx 180 ry 50 rz -21.45 deg; joints [-12.947, -46.989, 110.366, 133.844, 70.852, 108.856, -1868.548]
  MoveL 866 to (13.47, 311.83, 190) mm, rotated rx 180 ry 50 rz -14.57 deg; joints [-12.549, -46.948, 110.255, 134.226, 70.675, 108.778, -1875.435]
  MoveL 867 to (7.35, 312.92, 200) mm, rotated rx 180 ry 50 rz -7.9 deg; joints [-12.152, -46.9, 110.137, 134.607, 70.498, 108.698, -1882.098]
  MoveL 868 to (1.41, 313.37, 210) mm, rotated rx -180 ry 50 rz -1.51 deg; joints [-11.755, -46.845, 110.013, 134.989, 70.323, 108.616, -1888.487]
  MoveL 869 to (-4.24, 313.23, 220) mm, rotated rx 180 ry 50 rz 4.55 deg; joints [-11.359, -46.784, 109.883, 135.37, 70.147, 108.534, -1894.554]
  MoveL 870 to (-9.52, 312.61, 230) mm, rotated rx -180 ry 50 rz 10.25 deg; joints [-10.964, -46.717, 109.746, 135.75, 69.972, 108.45, -1900.254]
  MoveL 871 to (-14.35, 311.61, 240) mm, rotated rx 180 ry 50 rz 15.54 deg; joints [-10.57, -46.645, 109.602, 136.131, 69.796, 108.366, -1905.543]
  MoveL 872 to (-18.7, 310.34, 250) mm, rotated rx -180 ry 50 rz 20.38 deg; joints [-10.177, -46.569, 109.453, 136.51, 69.619, 108.282, -1910.381]
  MoveL 873 to (-22.53, 308.91, 260) mm, rotated rx -180 ry 50 rz 24.73 deg; joints [-9.784, -46.489, 109.297, 136.888, 69.441, 108.199, -1914.728]
  MoveL 874 to (-25.81, 307.44, 270) mm, rotated rx 180 ry 50 rz 28.55 deg; joints [-9.393, -46.406, 109.135, 137.265, 69.261, 108.116, -1918.548]
  MoveL 875 to (-28.54, 306.02, 280) mm, rotated rx -180 ry 50 rz 31.81 deg; joints [-9.003, -46.321, 108.967, 137.641, 69.079, 108.035, -1921.806]
  MoveL 876 to (-30.72, 304.75, 290) mm, rotated rx -180 ry 50 rz 34.47 deg; joints [-8.613, -46.233, 108.792, 138.015, 68.894, 107.955, -1924.467]
  MoveL 877 to (-58.22, 263.67, 290) mm, rotated rx -180 ry 50 rz 86.39 deg; joints [-8.613, -46.013, 108.776, 138.068, 69.046, 107.809, -1976.394]
  Set speed (60.0 mm/s)
  MoveL 878 to (-57.77, 266.15, 280) mm, rotated rx 180 ry 50 rz 83.92 deg; joints [-9.003, -46.106, 108.951, 137.692, 69.226, 107.891, -1973.924]
  MoveL 879 to (-57.08, 269.15, 270) mm, rotated rx 180 ry 50 rz 80.89 deg; joints [-9.393, -46.199, 109.12, 137.314, 69.402, 107.977, -1970.894]
  MoveL 880 to (-56.08, 272.6, 260) mm, rotated rx -180 ry 50 rz 77.33 deg; joints [-9.784, -46.292, 109.283, 136.935, 69.575, 108.065, -1967.333]
  MoveL 881 to (-54.69, 276.44, 250) mm, rotated rx 180 ry 50 rz 73.27 deg; joints [-10.177, -46.384, 109.439, 136.554, 69.744, 108.156, -1963.267]
  MoveL 882 to (-52.84, 280.57, 240) mm, rotated rx 180 ry 50 rz 68.72 deg; joints [-10.57, -46.474, 109.59, 136.171, 69.91, 108.249, -1958.724]
  MoveL 883 to (-50.46, 284.91, 230) mm, rotated rx 180 ry 50 rz 63.73 deg; joints [-10.964, -46.564, 109.735, 135.787, 70.074, 108.344, -1953.731]
  MoveL 884 to (-47.51, 289.33, 220) mm, rotated rx 180 ry 50 rz 58.32 deg; joints [-11.359, -46.651, 109.873, 135.401, 70.235, 108.441, -1948.316]
  MoveL 885 to (-43.95, 293.72, 210) mm, rotated rx 180 ry 50 rz 52.51 deg; joints [-11.755, -46.735, 110.005, 135.014, 70.395, 108.54, -1942.509]
  MoveL 886 to (-39.77, 297.95, 200) mm, rotated rx 180 ry 50 rz 46.34 deg; joints [-12.152, -46.816, 110.131, 134.627, 70.553, 108.639, -1936.342]
  MoveL 887 to (-34.96, 301.9, 190) mm, rotated rx 180 ry 50 rz 39.85 deg; joints [-12.549, -46.892, 110.251, 134.239, 70.711, 108.739, -1929.847]
  MoveL 888 to (-29.57, 305.43, 180) mm, rotated rx -180 ry 50 rz 33.06 deg; joints [-12.947, -46.964, 110.364, 133.85, 70.868, 108.838, -1923.063]
  MoveL 889 to (-23.65, 308.43, 170) mm, rotated rx -180 ry 50 rz 26.03 deg; joints [-13.346, -47.029, 110.471, 133.461, 71.026, 108.937, -1916.03]
  MoveL 890 to (-17.28, 310.79, 160) mm, rotated rx 180 ry 50 rz 18.79 deg; joints [-13.746, -47.089, 110.572, 133.072, 71.184, 109.035, -1908.791]
  MoveL 891 to (-10.57, 312.43, 150) mm, rotated rx -180 ry 50 rz 11.39 deg; joints [-14.146, -47.141, 110.666, 132.683, 71.343, 109.131, -1901.395]
  MoveL 892 to (-3.62, 313.27, 140) mm, rotated rx 180 ry 50 rz 3.89 deg; joints [-14.546, -47.186, 110.753, 132.294, 71.503, 109.225, -1893.889]
  MoveL 893 to (3.42, 313.28, 130) mm, rotated rx 180 ry 50 rz -3.67 deg; joints [-14.948, -47.223, 110.834, 131.906, 71.665, 109.317, -1886.327]
  MoveL 894 to (10.42, 312.45, 120) mm, rotated rx -180 ry 50 rz -11.24 deg; joints [-15.349, -47.253, 110.908, 131.518, 71.828, 109.407, -1878.761]
  MoveL 895 to (17.25, 310.8, 110) mm, rotated rx 180 ry 50 rz -18.76 deg; joints [-15.751, -47.275, 110.976, 131.13, 71.992, 109.495, -1871.243]
  MoveL 896 to (23.78, 308.38, 100) mm, rotated rx 180 ry 50 rz -26.18 deg; joints [-16.154, -47.29, 111.037, 130.743, 72.157, 109.58, -1863.825]
  MoveL 897 to (29.89, 305.25, 90) mm, rotated rx 180 ry 50 rz -33.45 deg; joints [-16.557, -47.298, 111.092, 130.355, 72.323, 109.665, -1856.554]
  MoveL 898 to (35.48, 301.51, 80) mm, rotated rx -180 ry 50 rz -40.52 deg; joints [-16.96, -47.3, 111.141, 129.968, 72.489, 109.748, -1849.477]
  MoveL 899 to (40.49, 297.28, 70) mm, rotated rx -180 ry 50 rz -47.36 deg; joints [-17.364, -47.296, 111.182, 129.581, 72.655, 109.83, -1842.636]
  MoveL 900 to (44.86, 292.68, 60) mm, rotated rx 180 ry 50 rz -53.93 deg; joints [-17.768, -47.287, 111.218, 129.194, 72.82, 109.913, -1836.069]
  MoveL 901 to (48.58, 287.83, 50) mm, rotated rx -180 ry 50 rz -60.19 deg; joints [-18.172, -47.275, 111.247, 128.807, 72.984, 109.995, -1829.813]
  MoveL 902 to (51.63, 282.88, 40) mm, rotated rx 180 ry 50 rz -66.1 deg; joints [-18.576, -47.259, 111.27, 128.419, 73.147, 110.079, -1823.9]
  MoveL 903 to (54.06, 277.94, 30) mm, rotated rx 180 ry 50 rz -71.64 deg; joints [-18.981, -47.241, 111.287, 128.031, 73.308, 110.165, -1818.36]
  MoveL 904 to (55.91, 273.13, 20) mm, rotated rx -180 ry 50 rz -76.78 deg; joints [-19.385, -47.221, 111.298, 127.642, 73.466, 110.253, -1813.221]
  MoveL 905 to (57.23, 268.56, 10) mm, rotated rx -180 ry 50 rz -81.49 deg; joints [-19.79, -47.199, 111.302, 127.252, 73.623, 110.343, -1808.51]
  MoveL 906 to (58.12, 264.32, 0) mm, rotated rx 180 ry 50 rz -85.75 deg; joints [-20.194, -47.176, 111.301, 126.862, 73.776, 110.437, -1804.254]
  MoveL 907 to (-58.22, 263.67, 290) mm, rotated rx 180 ry 50 rz 86.39 deg; joints [-8.613, -46.013, 108.776, 138.068, 69.046, 107.809, -1976.394]
  Set speed (60.0 mm/s)
  MoveL 908 to (-78.63, 259.66, 290) mm, rotated rx -180 ry 50 rz 90.25 deg; joints [-8.613, -44.905, 108.674, 138.32, 69.797, 107.092, -1980.245]
  MoveL 909 to (58.12, 264.32, 0) mm, rotated rx 180 ry 50 rz -85.75 deg; joints [-20.194, -47.176, 111.301, 126.862, 73.776, 110.437, -1804.254]
  Set speed (60.0 mm/s)
  MoveL 910 to (76.17, 274.65, 0) mm, rotated rx 180 ry 50 rz -79.11 deg; joints [-20.194, -46.096, 111.204, 127.086, 74.368, 109.619, -1810.889]
  MoveL 911 to (58.12, 264.32, 0) mm, rotated rx 180 ry 50 rz -85.75 deg; joints [-20.194, -47.176, 111.301, 126.862, 73.776, 110.437, -1804.254]
  Set speed (60.0 mm/s)
  MoveL 912 to (57.23, 268.56, 10) mm, rotated rx 180 ry 50 rz -81.49 deg; joints [-19.79, -47.199, 111.302, 127.252, 73.623, 110.343, -1808.51]
  MoveL 913 to (55.91, 273.13, 20) mm, rotated rx -180 ry 50 rz -76.78 deg; joints [-19.385, -47.221, 111.298, 127.642, 73.466, 110.253, -1813.221]
  MoveL 914 to (54.06, 277.94, 30) mm, rotated rx -180 ry 50 rz -71.64 deg; joints [-18.981, -47.241, 111.287, 128.031, 73.308, 110.165, -1818.36]
  MoveL 915 to (51.63, 282.88, 40) mm, rotated rx -180 ry 50 rz -66.1 deg; joints [-18.576, -47.259, 111.27, 128.419, 73.147, 110.079, -1823.9]
  MoveL 916 to (48.58, 287.83, 50) mm, rotated rx 180 ry 50 rz -60.19 deg; joints [-18.172, -47.275, 111.247, 128.807, 72.984, 109.995, -1829.813]
  MoveL 917 to (44.86, 292.68, 60) mm, rotated rx 180 ry 50 rz -53.93 deg; joints [-17.768, -47.287, 111.218, 129.194, 72.82, 109.913, -1836.069]
  MoveL 918 to (40.49, 297.28, 70) mm, rotated rx -180 ry 50 rz -47.36 deg; joints [-17.364, -47.296, 111.182, 129.581, 72.655, 109.83, -1842.636]
  MoveL 919 to (35.48, 301.51, 80) mm, rotated rx -180 ry 50 rz -40.52 deg; joints [-16.96, -47.3, 111.141, 129.968, 72.489, 109.748, -1849.477]
  MoveL 920 to (29.89, 305.25, 90) mm, rotated rx 180 ry 50 rz -33.45 deg; joints [-16.557, -47.298, 111.092, 130.355, 72.323, 109.665, -1856.554]
  MoveL 921 to (23.78, 308.38, 100) mm, rotated rx -180 ry 50 rz -26.18 deg; joints [-16.154, -47.29, 111.037, 130.743, 72.157, 109.58, -1863.825]
  MoveL 922 to (17.25, 310.8, 110) mm, rotated rx 180 ry 50 rz -18.76 deg; joints [-15.751, -47.275, 110.976, 131.13, 71.992, 109.495, -1871.243]
  MoveL 923 to (10.42, 312.45, 120) mm, rotated rx 180 ry 50 rz -11.24 deg; joints [-15.349, -47.253, 110.908, 131.518, 71.828, 109.407, -1878.761]
  MoveL 924 to (3.42, 313.28, 130) mm, rotated rx 180 ry 50 rz -3.67 deg; joints [-14.948, -47.223, 110.834, 131.906, 71.665, 109.317, -1886.327]
  MoveL 925 to (-3.62, 313.27, 140) mm, rotated rx -180 ry 50 rz 3.89 deg; joints [-14.546, -47.186, 110.753, 132.294, 71.503, 109.225, -1893.889]
  MoveL 926 to (-10.57, 312.43, 150) mm, rotated rx -180 ry 50 rz 11.39 deg; joints [-14.146, -47.141, 110.666, 132.683, 71.343, 109.131, -1901.395]
  MoveL 927 to (-17.28, 310.79, 160) mm, rotated rx -180 ry 50 rz 18.79 deg; joints [-13.746, -47.089, 110.572, 133.072, 71.184, 109.035, -1908.791]
  MoveL 928 to (-23.65, 308.43, 170) mm, rotated rx 180 ry 50 rz 26.03 deg; joints [-13.346, -47.029, 110.471, 133.461, 71.026, 108.937, -1916.03]
  MoveL 929 to (-29.57, 305.43, 180) mm, rotated rx -180 ry 50 rz 33.06 deg; joints [-12.947, -46.964, 110.364, 133.85, 70.868, 108.838, -1923.063]
  MoveL 930 to (-34.96, 301.9, 190) mm, rotated rx -180 ry 50 rz 39.85 deg; joints [-12.549, -46.892, 110.251, 134.239, 70.711, 108.739, -1929.847]
  MoveL 931 to (-39.77, 297.95, 200) mm, rotated rx 180 ry 50 rz 46.34 deg; joints [-12.152, -46.816, 110.131, 134.627, 70.553, 108.639, -1936.342]
  MoveL 932 to (-43.95, 293.72, 210) mm, rotated rx 180 ry 50 rz 52.51 deg; joints [-11.755, -46.735, 110.005, 135.014, 70.395, 108.54, -1942.509]
  MoveL 933 to (-47.51, 289.33, 220) mm, rotated rx 180 ry 50 rz 58.32 deg; joints [-11.359, -46.651, 109.873, 135.401, 70.235, 108.441, -1948.316]
  MoveL 934 to (-50.46, 284.91, 230) mm, rotated rx 180 ry 50 rz 63.73 deg; joints [-10.964, -46.564, 109.735, 135.787, 70.074, 108.344, -1953.731]
  MoveL 935 to (-52.84, 280.57, 240) mm, rotated rx 180 ry 50 rz 68.72 deg; joints [-10.57, -46.474, 109.59, 136.171, 69.91, 108.249, -1958.724]
  MoveL 936 to (-54.69, 276.44, 250) mm, rotated rx 180 ry 50 rz 73.27 deg; joints [-10.177, -46.384, 109.439, 136.554, 69.744, 108.156, -1963.267]
  MoveL 937 to (-56.08, 272.6, 260) mm, rotated rx -180 ry 50 rz 77.33 deg; joints [-9.784, -46.292, 109.283, 136.935, 69.575, 108.065, -1967.333]
  MoveL 938 to (-57.08, 269.15, 270) mm, rotated rx -180 ry 50 rz 80.89 deg; joints [-9.393, -46.199, 109.12, 137.314, 69.402, 107.977, -1970.894]
  MoveL 939 to (-57.77, 266.15, 280) mm, rotated rx 180 ry 50 rz 83.92 deg; joints [-9.003, -46.106, 108.951, 137.692, 69.226, 107.891, -1973.924]
  MoveL 940 to (-58.22, 263.67, 290) mm, rotated rx 180 ry 50 rz 86.39 deg; joints [-8.613, -46.013, 108.776, 138.068, 69.046, 107.809, -1976.394]
  MoveL 941 to (-78.63, 259.66, 290) mm, rotated rx -180 ry 50 rz 90.25 deg; joints [-8.613, -44.905, 108.674, 138.32, 69.797, 107.092, -1980.245]
  Set speed (60.0 mm/s)
  MoveL 942 to (-78.34, 263.02, 280) mm, rotated rx -180 ry 50 rz 87.79 deg; joints [-9.003, -44.996, 108.849, 137.944, 69.974, 107.169, -1977.792]
  MoveL 943 to (-77.78, 267.1, 270) mm, rotated rx -180 ry 50 rz 84.79 deg; joints [-9.393, -45.087, 109.019, 137.566, 70.147, 107.248, -1974.787]
  MoveL 944 to (-76.86, 271.82, 260) mm, rotated rx 180 ry 50 rz 81.26 deg; joints [-9.784, -45.178, 109.182, 137.187, 70.316, 107.331, -1971.259]
  MoveL 945 to (-75.48, 277.1, 250) mm, rotated rx 180 ry 50 rz 77.24 deg; joints [-10.177, -45.269, 109.339, 136.805, 70.482, 107.416, -1967.238]
  MoveL 946 to (-73.51, 282.82, 240) mm, rotated rx -180 ry 50 rz 72.75 deg; joints [-10.57, -45.359, 109.491, 136.423, 70.645, 107.503, -1962.753]
  MoveL 947 to (-70.88, 288.88, 230) mm, rotated rx -180 ry 50 rz 67.83 deg; joints [-10.964, -45.448, 109.636, 136.038, 70.805, 107.593, -1957.833]
  MoveL 948 to (-67.49, 295.12, 220) mm, rotated rx 180 ry 50 rz 62.51 deg; joints [-11.359, -45.534, 109.776, 135.652, 70.962, 107.685, -1952.509]
  MoveL 949 to (-63.28, 301.4, 210) mm, rotated rx 180 ry 50 rz 56.81 deg; joints [-11.755, -45.619, 109.909, 135.265, 71.118, 107.778, -1946.81]
  MoveL 950 to (-58.22, 307.54, 200) mm, rotated rx 180 ry 50 rz 50.77 deg; joints [-12.152, -45.7, 110.035, 134.877, 71.271, 107.873, -1940.77]
  MoveL 951 to (-52.31, 313.38, 190) mm, rotated rx 180 ry 50 rz 44.42 deg; joints [-12.549, -45.777, 110.156, 134.489, 71.424, 107.968, -1934.421]
  MoveL 952 to (-45.56, 318.73, 180) mm, rotated rx 180 ry 50 rz 37.8 deg; joints [-12.947, -45.85, 110.27, 134.099, 71.576, 108.063, -1927.8]
  MoveL 953 to (-38.04, 323.45, 170) mm, rotated rx 180 ry 50 rz 30.95 deg; joints [-13.346, -45.917, 110.378, 133.71, 71.728, 108.158, -1920.945]
  MoveL 954 to (-29.85, 327.37, 160) mm, rotated rx 180 ry 50 rz 23.9 deg; joints [-13.746, -45.978, 110.479, 133.32, 71.88, 108.253, -1913.897]
  MoveL 955 to (-21.11, 330.36, 150) mm, rotated rx -180 ry 50 rz 16.7 deg; joints [-14.146, -46.033, 110.573, 132.93, 72.033, 108.346, -1906.697]
  MoveL 956 to (-11.96, 332.32, 140) mm, rotated rx -180 ry 50 rz 9.39 deg; joints [-14.546, -46.08, 110.661, 132.54, 72.187, 108.437, -1899.391]
  MoveL 957 to (-2.59, 333.2, 130) mm, rotated rx 180 ry 50 rz 2.03 deg; joints [-14.948, -46.121, 110.742, 132.15, 72.342, 108.527, -1892.026]
  MoveL 958 to (6.83, 332.94, 120) mm, rotated rx -180 ry 50 rz -5.35 deg; joints [-15.349, -46.153, 110.817, 131.76, 72.498, 108.615, -1884.647]
  MoveL 959 to (16.13, 331.57, 110) mm, rotated rx -180 ry 50 rz -12.7 deg; joints [-15.751, -46.178, 110.885, 131.371, 72.655, 108.701, -1877.302]
  MoveL 960 to (25.11, 329.13, 100) mm, rotated rx 180 ry 50 rz -19.96 deg; joints [-16.154, -46.196, 110.946, 130.982, 72.813, 108.785, -1870.039]
  MoveL 961 to (33.62, 325.71, 90) mm, rotated rx -180 ry 50 rz -27.1 deg; joints [-16.557, -46.206, 111, 130.593, 72.972, 108.868, -1862.902]
  MoveL 962 to (41.52, 321.41, 80) mm, rotated rx 180 ry 50 rz -34.06 deg; joints [-16.96, -46.211, 111.048, 130.204, 73.131, 108.949, -1855.936]
  MoveL 963 to (48.7, 316.39, 70) mm, rotated rx 180 ry 50 rz -40.82 deg; joints [-17.364, -46.209, 111.09, 129.816, 73.29, 109.03, -1849.182]
  MoveL 964 to (55.08, 310.79, 60) mm, rotated rx 180 ry 50 rz -47.32 deg; joints [-17.768, -46.202, 111.125, 129.427, 73.448, 109.11, -1842.679]
  MoveL 965 to (60.61, 304.79, 50) mm, rotated rx -180 ry 50 rz -53.53 deg; joints [-18.172, -46.191, 111.154, 129.038, 73.606, 109.191, -1836.465]
  MoveL 966 to (65.29, 298.57, 40) mm, rotated rx 180 ry 50 rz -59.43 deg; joints [-18.576, -46.177, 111.176, 128.649, 73.762, 109.273, -1830.575]
  MoveL 967 to (69.12, 292.29, 30) mm, rotated rx -180 ry 50 rz -64.96 deg; joints [-18.981, -46.159, 111.192, 128.259, 73.917, 109.356, -1825.041]
  MoveL 968 to (72.16, 286.11, 20) mm, rotated rx 180 ry 50 rz -70.1 deg; joints [-19.385, -46.14, 111.202, 127.869, 74.07, 109.441, -1819.895]
  MoveL 969 to (74.48, 280.19, 10) mm, rotated rx 180 ry 50 rz -74.83 deg; joints [-19.79, -46.118, 111.206, 127.478, 74.22, 109.529, -1815.168]
  MoveL 970 to (76.17, 274.65, 0) mm, rotated rx 180 ry 50 rz -79.11 deg; joints [-20.194, -46.096, 111.204, 127.086, 74.368, 109.619, -1810.889]
  MoveL 971 to (-78.63, 259.66, 290) mm, rotated rx -180 ry 50 rz 90.25 deg; joints [-8.613, -44.905, 108.674, 138.32, 69.797, 107.092, -1980.245]
  Set speed (60.0 mm/s)
  MoveL 972 to (-58.93, 252.99, 290) mm, rotated rx 180 ry 50 rz 96.78 deg; joints [-8.613, -45.958, 108.772, 138.081, 69.084, 107.773, -1986.784]
  MoveL 973 to (76.17, 274.65, 0) mm, rotated rx 180 ry 50 rz -79.11 deg; joints [-20.194, -46.096, 111.204, 127.086, 74.368, 109.619, -1810.889]
  Set speed (60.0 mm/s)
  MoveL 974 to (55.37, 274.67, 0) mm, rotated rx 180 ry 50 rz -75.16 deg; joints [-20.194, -47.232, 111.305, 126.85, 73.745, 110.479, -1814.838]
  MoveL 975 to (76.17, 274.65, 0) mm, rotated rx 180 ry 50 rz -79.11 deg; joints [-20.194, -46.096, 111.204, 127.086, 74.368, 109.619, -1810.889]
  Set speed (60.0 mm/s)
  MoveL 976 to (74.48, 280.19, 10) mm, rotated rx 180 ry 50 rz -74.83 deg; joints [-19.79, -46.118, 111.206, 127.478, 74.22, 109.529, -1815.168]
  MoveL 977 to (72.16, 286.11, 20) mm, rotated rx 180 ry 50 rz -70.1 deg; joints [-19.385, -46.14, 111.202, 127.869, 74.07, 109.441, -1819.895]
  MoveL 978 to (69.12, 292.29, 30) mm, rotated rx -180 ry 50 rz -64.96 deg; joints [-18.981, -46.159, 111.192, 128.259, 73.917, 109.356, -1825.041]
  MoveL 979 to (65.29, 298.57, 40) mm, rotated rx -180 ry 50 rz -59.43 deg; joints [-18.576, -46.177, 111.176, 128.649, 73.762, 109.273, -1830.575]
  MoveL 980 to (60.61, 304.79, 50) mm, rotated rx 180 ry 50 rz -53.53 deg; joints [-18.172, -46.191, 111.154, 129.038, 73.606, 109.191, -1836.465]
  MoveL 981 to (55.08, 310.79, 60) mm, rotated rx -180 ry 50 rz -47.32 deg; joints [-17.768, -46.202, 111.125, 129.427, 73.448, 109.11, -1842.679]
  MoveL 982 to (48.7, 316.39, 70) mm, rotated rx 180 ry 50 rz -40.82 deg; joints [-17.364, -46.209, 111.09, 129.816, 73.29, 109.03, -1849.182]
  MoveL 983 to (41.52, 321.41, 80) mm, rotated rx -180 ry 50 rz -34.06 deg; joints [-16.96, -46.211, 111.048, 130.204, 73.131, 108.949, -1855.936]
  MoveL 984 to (33.62, 325.71, 90) mm, rotated rx -180 ry 50 rz -27.1 deg; joints [-16.557, -46.206, 111, 130.593, 72.972, 108.868, -1862.902]
  MoveL 985 to (25.11, 329.13, 100) mm, rotated rx 180 ry 50 rz -19.96 deg; joints [-16.154, -46.196, 110.946, 130.982, 72.813, 108.785, -1870.039]
  MoveL 986 to (16.13, 331.57, 110) mm, rotated rx 180 ry 50 rz -12.7 deg; joints [-15.751, -46.178, 110.885, 131.371, 72.655, 108.701, -1877.302]
  MoveL 987 to (6.83, 332.94, 120) mm, rotated rx -180 ry 50 rz -5.35 deg; joints [-15.349, -46.153, 110.817, 131.76, 72.498, 108.615, -1884.647]
  MoveL 988 to (-2.59, 333.2, 130) mm, rotated rx -180 ry 50 rz 2.03 deg; joints [-14.948, -46.121, 110.742, 132.15, 72.342, 108.527, -1892.026]
  MoveL 989 to (-11.96, 332.32, 140) mm, rotated rx 180 ry 50 rz 9.39 deg; joints [-14.546, -46.08, 110.661, 132.54, 72.187, 108.437, -1899.391]
  MoveL 990 to (-21.11, 330.36, 150) mm, rotated rx 180 ry 50 rz 16.7 deg; joints [-14.146, -46.033, 110.573, 132.93, 72.033, 108.346, -1906.697]
  MoveL 991 to (-29.85, 327.37, 160) mm, rotated rx -180 ry 50 rz 23.9 deg; joints [-13.746, -45.978, 110.479, 133.32, 71.88, 108.253, -1913.897]
  MoveL 992 to (-38.04, 323.45, 170) mm, rotated rx 180 ry 50 rz 30.95 deg; joints [-13.346, -45.917, 110.378, 133.71, 71.728, 108.158, -1920.945]
  MoveL 993 to (-45.56, 318.73, 180) mm, rotated rx -180 ry 50 rz 37.8 deg; joints [-12.947, -45.85, 110.27, 134.099, 71.576, 108.063, -1927.8]
  MoveL 994 to (-52.31, 313.38, 190) mm, rotated rx 180 ry 50 rz 44.42 deg; joints [-12.549, -45.777, 110.156, 134.489, 71.424, 107.968, -1934.421]
  MoveL 995 to (-58.22, 307.54, 200) mm, rotated rx 180 ry 50 rz 50.77 deg; joints [-12.152, -45.7, 110.035, 134.877, 71.271, 107.873, -1940.77]
  MoveL 996 to (-63.28, 301.4, 210) mm, rotated rx 180 ry 50 rz 56.81 deg; joints [-11.755, -45.619, 109.909, 135.265, 71.118, 107.778, -1946.81]
  MoveL 997 to (-67.49, 295.12, 220) mm, rotated rx 180 ry 50 rz 62.51 deg; joints [-11.359, -45.534, 109.776, 135.652, 70.962, 107.685, -1952.509]
  MoveL 998 to (-70.88, 288.88, 230) mm, rotated rx 180 ry 50 rz 67.83 deg; joints [-10.964, -45.448, 109.636, 136.038, 70.805, 107.593, -1957.833]
  MoveL 999 to (-73.51, 282.82, 240) mm, rotated rx -180 ry 50 rz 72.75 deg; joints [-10.57, -45.359, 109.491, 136.423, 70.645, 107.503, -1962.753]
  MoveL 1000 to (-75.48, 277.1, 250) mm, rotated rx -180 ry 50 rz 77.24 deg; joints [-10.177, -45.269, 109.339, 136.805, 70.482, 107.416, -1967.238]
  MoveL 1001 to (-76.86, 271.82, 260) mm, rotated rx -180 ry 50 rz 81.26 deg; joints [-9.784, -45.178, 109.182, 137.187, 70.316, 107.331, -1971.259]
  MoveL 1002 to (-77.78, 267.1, 270) mm, rotated rx 180 ry 50 rz 84.79 deg; joints [-9.393, -45.087, 109.019, 137.566, 70.147, 107.248, -1974.787]
  MoveL 1003 to (-78.34, 263.02, 280) mm, rotated rx -180 ry 50 rz 87.79 deg; joints [-9.003, -44.996, 108.849, 137.944, 69.974, 107.169, -1977.792]
  MoveL 1004 to (-78.63, 259.66, 290) mm, rotated rx -180 ry 50 rz 90.25 deg; joints [-8.613, -44.905, 108.674, 138.32, 69.797, 107.092, -1980.245]
  MoveL 1005 to (-58.93, 252.99, 290) mm, rotated rx 180 ry 50 rz 96.78 deg; joints [-8.613, -45.958, 108.772, 138.081, 69.084, 107.773, -1986.784]
  Set speed (60.0 mm/s)
  MoveL 1006 to (-58.94, 255.51, 280) mm, rotated rx 180 ry 50 rz 94.36 deg; joints [-9.003, -46.051, 108.947, 137.705, 69.264, 107.855, -1984.356]
  MoveL 1007 to (-58.8, 258.59, 270) mm, rotated rx 180 ry 50 rz 91.38 deg; joints [-9.393, -46.144, 109.115, 137.327, 69.44, 107.94, -1981.378]
  MoveL 1008 to (-58.44, 262.16, 260) mm, rotated rx -180 ry 50 rz 87.88 deg; joints [-9.784, -46.237, 109.278, 136.948, 69.612, 108.028, -1977.879]
  MoveL 1009 to (-57.77, 266.19, 250) mm, rotated rx 180 ry 50 rz 83.88 deg; joints [-10.177, -46.329, 109.435, 136.566, 69.781, 108.119, -1973.884]
  MoveL 1010 to (-56.69, 270.59, 240) mm, rotated rx 180 ry 50 rz 79.42 deg; joints [-10.57, -46.421, 109.586, 136.183, 69.946, 108.213, -1969.42]
  MoveL 1011 to (-55.14, 275.28, 230) mm, rotated rx 180 ry 50 rz 74.51 deg; joints [-10.964, -46.512, 109.731, 135.799, 70.108, 108.309, -1964.512]
  MoveL 1012 to (-53.04, 280.16, 220) mm, rotated rx 180 ry 50 rz 69.19 deg; joints [-11.359, -46.601, 109.87, 135.413, 70.268, 108.407, -1959.189]
  MoveL 1013 to (-50.33, 285.12, 210) mm, rotated rx -180 ry 50 rz 63.48 deg; joints [-11.755, -46.688, 110.002, 135.025, 70.426, 108.507, -1953.477]
  MoveL 1014 to (-46.98, 290.04, 200) mm, rotated rx 180 ry 50 rz 57.4 deg; joints [-12.152, -46.772, 110.128, 134.637, 70.582, 108.608, -1947.405]
  MoveL 1015 to (-42.97, 294.79, 190) mm, rotated rx 180 ry 50 rz 51 deg; joints [-12.549, -46.852, 110.248, 134.248, 70.737, 108.711, -1941.005]
  MoveL 1016 to (-38.31, 299.24, 180) mm, rotated rx 180 ry 50 rz 44.31 deg; joints [-12.947, -46.929, 110.362, 133.858, 70.891, 108.813, -1934.31]
  MoveL 1017 to (-33.03, 303.26, 170) mm, rotated rx -180 ry 50 rz 37.36 deg; joints [-13.346, -47, 110.469, 133.468, 71.045, 108.916, -1927.357]
  MoveL 1018 to (-27.19, 306.74, 160) mm, rotated rx -180 ry 50 rz 30.19 deg; joints [-13.746, -47.066, 110.57, 133.077, 71.199, 109.018, -1920.187]
  MoveL 1019 to (-20.88, 309.56, 150) mm, rotated rx 180 ry 50 rz 22.84 deg; joints [-14.146, -47.125, 110.665, 132.687, 71.353, 109.119, -1912.844]
  MoveL 1020 to (-14.2, 311.65, 140) mm, rotated rx 180 ry 50 rz 15.37 deg; joints [-14.546, -47.177, 110.752, 132.296, 71.509, 109.218, -1905.374]
  MoveL 1021 to (-7.28, 312.93, 130) mm, rotated rx 180 ry 50 rz 7.83 deg; joints [-14.948, -47.221, 110.834, 131.906, 71.666, 109.316, -1897.828]
  MoveL 1022 to (-0.24, 313.38, 120) mm, rotated rx 180 ry 50 rz 0.26 deg; joints [-15.349, -47.258, 110.909, 131.517, 71.824, 109.411, -1890.258]
  MoveL 1023 to (6.77, 312.99, 110) mm, rotated rx 180 ry 50 rz -7.29 deg; joints [-15.751, -47.288, 110.977, 131.127, 71.984, 109.504, -1882.715]
  MoveL 1024 to (13.63, 311.79, 100) mm, rotated rx 180 ry 50 rz -14.75 deg; joints [-16.154, -47.31, 111.039, 130.738, 72.145, 109.595, -1875.252]
  MoveL 1025 to (20.21, 309.81, 90) mm, rotated rx -180 ry 50 rz -22.08 deg; joints [-16.557, -47.324, 111.094, 130.35, 72.307, 109.684, -1867.921]
  MoveL 1026 to (26.38, 307.15, 80) mm, rotated rx 180 ry 50 rz -29.23 deg; joints [-16.96, -47.332, 111.143, 129.961, 72.47, 109.772, -1860.769]
  MoveL 1027 to (32.08, 303.89, 70) mm, rotated rx 180 ry 50 rz -36.16 deg; joints [-17.364, -47.333, 111.185, 129.573, 72.632, 109.858, -1853.843]
  MoveL 1028 to (37.21, 300.16, 60) mm, rotated rx 180 ry 50 rz -42.82 deg; joints [-17.768, -47.329, 111.221, 129.185, 72.795, 109.944, -1847.185]
  MoveL 1029 to (41.73, 296.07, 50) mm, rotated rx 180 ry 50 rz -49.17 deg; joints [-18.172, -47.321, 111.251, 128.797, 72.957, 110.03, -1840.833]
  MoveL 1030 to (45.64, 291.75, 40) mm, rotated rx -180 ry 50 rz -55.18 deg; joints [-18.576, -47.308, 111.274, 128.408, 73.119, 110.117, -1834.824]
  MoveL 1031 to (48.92, 287.33, 30) mm, rotated rx 180 ry 50 rz -60.81 deg; joints [-18.981, -47.292, 111.291, 128.02, 73.278, 110.204, -1829.19]
  MoveL 1032 to (51.6, 282.93, 20) mm, rotated rx 180 ry 50 rz -66.04 deg; joints [-19.385, -47.274, 111.302, 127.63, 73.436, 110.294, -1823.962]
  MoveL 1033 to (53.73, 278.68, 10) mm, rotated rx -180 ry 50 rz -70.83 deg; joints [-19.79, -47.253, 111.306, 127.241, 73.592, 110.385, -1819.169]
  MoveL 1034 to (55.37, 274.67, 0) mm, rotated rx 180 ry 50 rz -75.16 deg; joints [-20.194, -47.232, 111.305, 126.85, 73.745, 110.479, -1814.838]
  MoveL 1035 to (-58.93, 252.99, 290) mm, rotated rx -180 ry 50 rz 96.78 deg; joints [-8.613, -45.958, 108.772, 138.081, 69.084, 107.773, -1986.784]
  Set speed (60.0 mm/s)
  MoveL 1036 to (-37.11, 208.63, 290) mm, rotated rx 180 ry 50 rz 144.16 deg; joints [-8.613, -45.739, 108.754, 138.132, 69.233, 107.629, -2034.156]
  MoveL 1037 to (55.37, 274.67, 0) mm, rotated rx 180 ry 50 rz -75.16 deg; joints [-20.194, -47.232, 111.305, 126.85, 73.745, 110.479, -2174.838]
  Set speed (60.0 mm/s)
  MoveL 1038 to (20.49, 309.71, 0) mm, rotated rx -180 ry 50 rz -22.4 deg; joints [-20.194, -47.427, 111.319, 126.808, 73.637, 110.631, -2227.595]
  MoveL 1039 to (55.37, 274.67, 0) mm, rotated rx 180 ry 50 rz -75.16 deg; joints [-20.194, -47.232, 111.305, 126.85, 73.745, 110.479, -2174.838]
  Set speed (60.0 mm/s)
  MoveL 1040 to (53.73, 278.68, 10) mm, rotated rx 180 ry 50 rz -70.83 deg; joints [-19.79, -47.253, 111.306, 127.241, 73.592, 110.385, -2179.169]
  MoveL 1041 to (51.6, 282.93, 20) mm, rotated rx 180 ry 50 rz -66.04 deg; joints [-19.385, -47.274, 111.302, 127.63, 73.436, 110.294, -2183.962]
  MoveL 1042 to (48.92, 287.33, 30) mm, rotated rx 180 ry 50 rz -60.81 deg; joints [-18.981, -47.292, 111.291, 128.02, 73.278, 110.204, -2189.19]
  MoveL 1043 to (45.64, 291.75, 40) mm, rotated rx 180 ry 50 rz -55.18 deg; joints [-18.576, -47.308, 111.274, 128.408, 73.119, 110.117, -2194.824]
  MoveL 1044 to (41.73, 296.07, 50) mm, rotated rx 180 ry 50 rz -49.17 deg; joints [-18.172, -47.321, 111.251, 128.797, 72.957, 110.03, -2200.833]
  MoveL 1045 to (37.21, 300.16, 60) mm, rotated rx -180 ry 50 rz -42.82 deg; joints [-17.768, -47.329, 111.221, 129.185, 72.795, 109.944, -2207.185]
  MoveL 1046 to (32.08, 303.89, 70) mm, rotated rx 180 ry 50 rz -36.16 deg; joints [-17.364, -47.333, 111.185, 129.573, 72.632, 109.858, -2213.843]
  MoveL 1047 to (26.38, 307.15, 80) mm, rotated rx 180 ry 50 rz -29.23 deg; joints [-16.96, -47.332, 111.143, 129.961, 72.47, 109.772, -2220.769]
  MoveL 1048 to (20.21, 309.81, 90) mm, rotated rx 180 ry 50 rz -22.08 deg; joints [-16.557, -47.324, 111.094, 130.35, 72.307, 109.684, -2227.921]
  MoveL 1049 to (13.63, 311.79, 100) mm, rotated rx -180 ry 50 rz -14.75 deg; joints [-16.154, -47.31, 111.039, 130.738, 72.145, 109.595, -2235.252]
  MoveL 1050 to (6.77, 312.99, 110) mm, rotated rx -180 ry 50 rz -7.29 deg; joints [-15.751, -47.288, 110.977, 131.127, 71.984, 109.504, -2242.715]
  MoveL 1051 to (-0.24, 313.38, 120) mm, rotated rx -180 ry 50 rz 0.26 deg; joints [-15.349, -47.258, 110.909, 131.517, 71.824, 109.411, -2250.258]
  MoveL 1052 to (-7.28, 312.93, 130) mm, rotated rx -180 ry 50 rz 7.83 deg; joints [-14.948, -47.221, 110.834, 131.906, 71.666, 109.316, -2257.828]
  MoveL 1053 to (-14.2, 311.65, 140) mm, rotated rx 180 ry 50 rz 15.37 deg; joints [-14.546, -47.177, 110.752, 132.296, 71.509, 109.218, -2265.374]
  MoveL 1054 to (-20.88, 309.56, 150) mm, rotated rx 180 ry 50 rz 22.84 deg; joints [-14.146, -47.125, 110.665, 132.687, 71.353, 109.119, -2272.844]
  MoveL 1055 to (-27.19, 306.74, 160) mm, rotated rx 180 ry 50 rz 30.19 deg; joints [-13.746, -47.066, 110.57, 133.077, 71.199, 109.018, -2280.187]
  MoveL 1056 to (-33.03, 303.26, 170) mm, rotated rx 180 ry 50 rz 37.36 deg; joints [-13.346, -47, 110.469, 133.468, 71.045, 108.916, -2287.357]
  MoveL 1057 to (-38.31, 299.24, 180) mm, rotated rx -180 ry 50 rz 44.31 deg; joints [-12.947, -46.929, 110.362, 133.858, 70.891, 108.813, -2294.31]
  MoveL 1058 to (-42.97, 294.79, 190) mm, rotated rx 180 ry 50 rz 51 deg; joints [-12.549, -46.852, 110.248, 134.248, 70.737, 108.711, -2301.005]
  MoveL 1059 to (-46.98, 290.04, 200) mm, rotated rx -180 ry 50 rz 57.4 deg; joints [-12.152, -46.772, 110.128, 134.637, 70.582, 108.608, -2307.405]
  MoveL 1060 to (-50.33, 285.12, 210) mm, rotated rx 180 ry 50 rz 63.48 deg; joints [-11.755, -46.688, 110.002, 135.025, 70.426, 108.507, -2313.477]
  MoveL 1061 to (-53.04, 280.16, 220) mm, rotated rx 180 ry 50 rz 69.19 deg; joints [-11.359, -46.601, 109.87, 135.413, 70.268, 108.407, -2319.189]
  MoveL 1062 to (-55.14, 275.28, 230) mm, rotated rx -180 ry 50 rz 74.51 deg; joints [-10.964, -46.512, 109.731, 135.799, 70.108, 108.309, -2324.512]
  MoveL 1063 to (-56.69, 270.59, 240) mm, rotated rx 180 ry 50 rz 79.42 deg; joints [-10.57, -46.421, 109.586, 136.183, 69.946, 108.213, -2329.42]
  MoveL 1064 to (-57.77, 266.19, 250) mm, rotated rx 180 ry 50 rz 83.88 deg; joints [-10.177, -46.329, 109.435, 136.566, 69.781, 108.119, -2333.884]
  MoveL 1065 to (-58.44, 262.16, 260) mm, rotated rx 180 ry 50 rz 87.88 deg; joints [-9.784, -46.237, 109.278, 136.948, 69.612, 108.028, -2337.879]
  MoveL 1066 to (-58.8, 258.59, 270) mm, rotated rx -180 ry 50 rz 91.38 deg; joints [-9.393, -46.144, 109.115, 137.327, 69.44, 107.94, -2341.378]
  MoveL 1067 to (-58.94, 255.51, 280) mm, rotated rx -180 ry 50 rz 94.36 deg; joints [-9.003, -46.051, 108.947, 137.705, 69.264, 107.855, -2344.356]
  MoveL 1068 to (-58.93, 252.99, 290) mm, rotated rx -180 ry 50 rz 96.78 deg; joints [-8.613, -45.958, 108.772, 138.081, 69.084, 107.773, -2346.784]
  MoveL 1069 to (-37.11, 208.63, 290) mm, rotated rx 180 ry 50 rz 144.16 deg; joints [-8.613, -45.739, 108.754, 138.132, 69.233, 107.629, -2394.156]
  Set speed (60.0 mm/s)
  MoveL 1070 to (-39.03, 210.26, 280) mm, rotated rx 180 ry 50 rz 141.88 deg; joints [-9.003, -45.827, 108.928, 137.757, 69.416, 107.707, -2391.877]
  MoveL 1071 to (-41.29, 212.35, 270) mm, rotated rx 180 ry 50 rz 139.09 deg; joints [-9.393, -45.914, 109.097, 137.381, 69.595, 107.787, -2389.089]
  MoveL 1072 to (-43.78, 214.95, 260) mm, rotated rx -180 ry 50 rz 135.82 deg; joints [-9.784, -46, 109.259, 137.003, 69.771, 107.87, -2385.82]
  MoveL 1073 to (-46.4, 218.08, 250) mm, rotated rx 180 ry 50 rz 132.1 deg; joints [-10.177, -46.087, 109.416, 136.623, 69.943, 107.955, -2382.097]
  MoveL 1074 to (-49.06, 221.75, 240) mm, rotated rx 180 ry 50 rz 127.95 deg; joints [-10.57, -46.173, 109.567, 136.241, 70.111, 108.044, -2377.947]
  MoveL 1075 to (-51.62, 225.97, 230) mm, rotated rx 180 ry 50 rz 123.4 deg; joints [-10.964, -46.259, 109.711, 135.857, 70.276, 108.136, -2373.396]
  MoveL 1076 to (-53.98, 230.73, 220) mm, rotated rx -180 ry 50 rz 118.47 deg; joints [-11.359, -46.345, 109.85, 135.472, 70.436, 108.231, -2368.469]
  MoveL 1077 to (-56, 236.01, 210) mm, rotated rx -180 ry 50 rz 113.19 deg; joints [-11.755, -46.431, 109.982, 135.085, 70.593, 108.329, -2363.192]
  MoveL 1078 to (-57.57, 241.75, 200) mm, rotated rx 180 ry 50 rz 107.59 deg; joints [-12.152, -46.517, 110.109, 134.696, 70.747, 108.431, -2357.589]
  MoveL 1079 to (-58.59, 247.88, 190) mm, rotated rx 180 ry 50 rz 101.68 deg; joints [-12.549, -46.603, 110.23, 134.305, 70.898, 108.536, -2351.684]
  MoveL 1080 to (-58.95, 254.32, 180) mm, rotated rx -180 ry 50 rz 95.5 deg; joints [-12.947, -46.687, 110.344, 133.914, 71.046, 108.643, -2345.504]
  MoveL 1081 to (-58.59, 260.95, 170) mm, rotated rx -180 ry 50 rz 89.07 deg; joints [-13.346, -46.77, 110.452, 133.521, 71.191, 108.753, -2339.073]
  MoveL 1082 to (-57.45, 267.65, 160) mm, rotated rx -180 ry 50 rz 82.42 deg; joints [-13.746, -46.851, 110.555, 133.126, 71.334, 108.865, -2332.419]
  MoveL 1083 to (-55.51, 274.28, 150) mm, rotated rx 180 ry 50 rz 75.57 deg; joints [-14.146, -46.929, 110.65, 132.732, 71.476, 108.978, -2325.573]
  MoveL 1084 to (-52.77, 280.72, 140) mm, rotated rx 180 ry 50 rz 68.57 deg; joints [-14.546, -47.004, 110.74, 132.336, 71.617, 109.093, -2318.565]
  MoveL 1085 to (-49.26, 286.82, 130) mm, rotated rx 180 ry 50 rz 61.43 deg; joints [-14.948, -47.075, 110.823, 131.94, 71.757, 109.209, -2311.431]
  MoveL 1086 to (-45.04, 292.47, 120) mm, rotated rx 180 ry 50 rz 54.21 deg; joints [-15.349, -47.14, 110.9, 131.543, 71.897, 109.324, -2304.209]
  MoveL 1087 to (-40.19, 297.56, 110) mm, rotated rx 180 ry 50 rz 46.94 deg; joints [-15.751, -47.2, 110.971, 131.147, 72.038, 109.439, -2296.94]
  MoveL 1088 to (-34.83, 302, 100) mm, rotated rx 180 ry 50 rz 39.67 deg; joints [-16.154, -47.254, 111.035, 130.751, 72.179, 109.554, -2289.668]
  MoveL 1089 to (-29.06, 305.72, 90) mm, rotated rx 180 ry 50 rz 32.44 deg; joints [-16.557, -47.301, 111.092, 130.355, 72.321, 109.667, -2282.441]
  MoveL 1090 to (-23.03, 308.7, 80) mm, rotated rx -180 ry 50 rz 25.31 deg; joints [-16.96, -47.341, 111.143, 129.959, 72.464, 109.778, -2275.308]
  MoveL 1091 to (-16.86, 310.92, 70) mm, rotated rx -180 ry 50 rz 18.32 deg; joints [-17.364, -47.373, 111.188, 129.564, 72.609, 109.888, -2268.32]
  MoveL 1092 to (-10.69, 312.41, 60) mm, rotated rx -180 ry 50 rz 11.53 deg; joints [-17.768, -47.399, 111.226, 129.169, 72.754, 109.997, -2261.529]
  MoveL 1093 to (-4.64, 313.2, 50) mm, rotated rx -180 ry 50 rz 4.98 deg; joints [-18.172, -47.418, 111.257, 128.775, 72.901, 110.104, -2254.983]
  MoveL 1094 to (1.18, 313.37, 40) mm, rotated rx 180 ry 50 rz -1.27 deg; joints [-18.576, -47.431, 111.282, 128.381, 73.048, 110.21, -2248.733]
  MoveL 1095 to (6.67, 313.01, 30) mm, rotated rx 180 ry 50 rz -7.17 deg; joints [-18.981, -47.437, 111.301, 127.988, 73.195, 110.315, -2242.826]
  MoveL 1096 to (11.76, 312.2, 20) mm, rotated rx 180 ry 50 rz -12.69 deg; joints [-19.385, -47.438, 111.313, 127.594, 73.343, 110.42, -2237.306]
  MoveL 1097 to (16.38, 311.06, 10) mm, rotated rx 180 ry 50 rz -17.78 deg; joints [-19.79, -47.435, 111.319, 127.201, 73.49, 110.525, -2232.216]
  MoveL 1098 to (20.49, 309.71, 0) mm, rotated rx 180 ry 50 rz -22.4 deg; joints [-20.194, -47.427, 111.319, 126.808, 73.637, 110.631, -2227.595]
  MoveL 1099 to (-37.11, 208.63, 290) mm, rotated rx 180 ry 50 rz 144.16 deg; joints [-8.613, -45.739, 108.754, 138.132, 69.233, 107.629, -2394.156]
  Set speed (60.0 mm/s)
  MoveL 1100 to (-43.85, 188.95, 290) mm, rotated rx 180 ry 50 rz 148.32 deg; joints [-8.613, -44.637, 108.645, 138.378, 69.974, 106.924, -2398.321]
  MoveL 1101 to (20.49, 309.71, 0) mm, rotated rx -180 ry 50 rz -22.4 deg; joints [-20.194, -47.427, 111.319, 126.808, 73.637, 110.631, -2227.595]
  Set speed (60.0 mm/s)
  MoveL 1102 to (20.57, 330.51, 0) mm, rotated rx -180 ry 50 rz -16.27 deg; joints [-20.194, -46.328, 111.227, 127.04, 74.242, 109.792, -2233.733]
  MoveL 1103 to (20.49, 309.71, 0) mm, rotated rx -180 ry 50 rz -22.4 deg; joints [-20.194, -47.427, 111.319, 126.808, 73.637, 110.631, -2227.595]
  Set speed (60.0 mm/s)
  MoveL 1104 to (16.38, 311.06, 10) mm, rotated rx -180 ry 50 rz -17.78 deg; joints [-19.79, -47.435, 111.319, 127.201, 73.49, 110.525, -2232.216]
  MoveL 1105 to (11.76, 312.2, 20) mm, rotated rx 180 ry 50 rz -12.69 deg; joints [-19.385, -47.438, 111.313, 127.594, 73.343, 110.42, -2237.306]
  MoveL 1106 to (6.67, 313.01, 30) mm, rotated rx -180 ry 50 rz -7.17 deg; joints [-18.981, -47.437, 111.301, 127.988, 73.195, 110.315, -2242.826]
  MoveL 1107 to (1.18, 313.37, 40) mm, rotated rx 180 ry 50 rz -1.27 deg; joints [-18.576, -47.431, 111.282, 128.381, 73.048, 110.21, -2248.733]
  MoveL 1108 to (-4.64, 313.2, 50) mm, rotated rx 180 ry 50 rz 4.98 deg; joints [-18.172, -47.418, 111.257, 128.775, 72.901, 110.104, -2254.983]
  MoveL 1109 to (-10.69, 312.41, 60) mm, rotated rx -180 ry 50 rz 11.53 deg; joints [-17.768, -47.399, 111.226, 129.169, 72.754, 109.997, -2261.529]
  MoveL 1110 to (-16.86, 310.92, 70) mm, rotated rx -180 ry 50 rz 18.32 deg; joints [-17.364, -47.373, 111.188, 129.564, 72.609, 109.888, -2268.32]
  MoveL 1111 to (-23.03, 308.7, 80) mm, rotated rx -180 ry 50 rz 25.31 deg; joints [-16.96, -47.341, 111.143, 129.959, 72.464, 109.778, -2275.308]
  MoveL 1112 to (-29.06, 305.72, 90) mm, rotated rx -180 ry 50 rz 32.44 deg; joints [-16.557, -47.301, 111.092, 130.355, 72.321, 109.667, -2282.441]
  MoveL 1113 to (-34.83, 302, 100) mm, rotated rx 180 ry 50 rz 39.67 deg; joints [-16.154, -47.254, 111.035, 130.751, 72.179, 109.554, -2289.668]
  MoveL 1114 to (-40.19, 297.56, 110) mm, rotated rx 180 ry 50 rz 46.94 deg; joints [-15.751, -47.2, 110.971, 131.147, 72.038, 109.439, -2296.94]
  MoveL 1115 to (-45.04, 292.47, 120) mm, rotated rx -180 ry 50 rz 54.21 deg; joints [-15.349, -47.14, 110.9, 131.543, 71.897, 109.324, -2304.209]
  MoveL 1116 to (-49.26, 286.82, 130) mm, rotated rx 180 ry 50 rz 61.43 deg; joints [-14.948, -47.075, 110.823, 131.94, 71.757, 109.209, -2311.431]
  MoveL 1117 to (-52.77, 280.72, 140) mm, rotated rx 180 ry 50 rz 68.57 deg; joints [-14.546, -47.004, 110.74, 132.336, 71.617, 109.093, -2318.565]
  MoveL 1118 to (-55.51, 274.28, 150) mm, rotated rx 180 ry 50 rz 75.57 deg; joints [-14.146, -46.929, 110.65, 132.732, 71.476, 108.978, -2325.573]
  MoveL 1119 to (-57.45, 267.65, 160) mm, rotated rx 180 ry 50 rz 82.42 deg; joints [-13.746, -46.851, 110.555, 133.126, 71.334, 108.865, -2332.419]
  MoveL 1120 to (-58.59, 260.95, 170) mm, rotated rx -180 ry 50 rz 89.07 deg; joints [-13.346, -46.77, 110.452, 133.521, 71.191, 108.753, -2339.073]
  MoveL 1121 to (-58.95, 254.32, 180) mm, rotated rx -180 ry 50 rz 95.5 deg; joints [-12.947, -46.687, 110.344, 133.914, 71.046, 108.643, -2345.504]
  MoveL 1122 to (-58.59, 247.88, 190) mm, rotated rx -180 ry 50 rz 101.68 deg; joints [-12.549, -46.603, 110.23, 134.305, 70.898, 108.536, -2351.684]
  MoveL 1123 to (-57.57, 241.75, 200) mm, rotated rx 180 ry 50 rz 107.59 deg; joints [-12.152, -46.517, 110.109, 134.696, 70.747, 108.431, -2357.589]
  MoveL 1124 to (-56, 236.01, 210) mm, rotated rx 180 ry 50 rz 113.19 deg; joints [-11.755, -46.431, 109.982, 135.085, 70.593, 108.329, -2363.192]
  MoveL 1125 to (-53.98, 230.73, 220) mm, rotated rx -180 ry 50 rz 118.47 deg; joints [-11.359, -46.345, 109.85, 135.472, 70.436, 108.231, -2368.469]
  MoveL 1126 to (-51.62, 225.97, 230) mm, rotated rx 180 ry 50 rz 123.4 deg; joints [-10.964, -46.259, 109.711, 135.857, 70.276, 108.136, -2373.396]
  MoveL 1127 to (-49.06, 221.75, 240) mm, rotated rx -180 ry 50 rz 127.95 deg; joints [-10.57, -46.173, 109.567, 136.241, 70.111, 108.044, -2377.947]
  MoveL 1128 to (-46.4, 218.08, 250) mm, rotated rx 180 ry 50 rz 132.1 deg; joints [-10.177, -46.087, 109.416, 136.623, 69.943, 107.955, -2382.097]
  MoveL 1129 to (-43.78, 214.95, 260) mm, rotated rx 180 ry 50 rz 135.82 deg; joints [-9.784, -46, 109.259, 137.003, 69.771, 107.87, -2385.82]
  MoveL 1130 to (-41.29, 212.35, 270) mm, rotated rx 180 ry 50 rz 139.09 deg; joints [-9.393, -45.914, 109.097, 137.381, 69.595, 107.787, -2389.089]
  MoveL 1131 to (-39.03, 210.26, 280) mm, rotated rx -180 ry 50 rz 141.88 deg; joints [-9.003, -45.827, 108.928, 137.757, 69.416, 107.707, -2391.877]
  MoveL 1132 to (-37.11, 208.63, 290) mm, rotated rx 180 ry 50 rz 144.16 deg; joints [-8.613, -45.739, 108.754, 138.132, 69.233, 107.629, -2394.156]
  MoveL 1133 to (-43.85, 188.95, 290) mm, rotated rx 180 ry 50 rz 148.32 deg; joints [-8.613, -44.637, 108.645, 138.378, 69.974, 106.924, -2398.321]
  Set speed (60.0 mm/s)
  MoveL 1134 to (-46.6, 190.89, 280) mm, rotated rx -180 ry 50 rz 146.01 deg; joints [-9.003, -44.722, 108.819, 138.003, 70.155, 106.995, -2396.008]
  MoveL 1135 to (-49.86, 193.4, 270) mm, rotated rx 180 ry 50 rz 143.18 deg; joints [-9.393, -44.806, 108.988, 137.627, 70.332, 107.069, -2393.179]
  MoveL 1136 to (-53.49, 196.56, 260) mm, rotated rx -180 ry 50 rz 139.86 deg; joints [-9.784, -44.89, 109.151, 137.249, 70.505, 107.145, -2389.865]
  MoveL 1137 to (-57.36, 200.4, 250) mm, rotated rx 180 ry 50 rz 136.1 deg; joints [-10.177, -44.974, 109.308, 136.869, 70.674, 107.224, -2386.095]
  MoveL 1138 to (-61.34, 204.96, 240) mm, rotated rx -180 ry 50 rz 131.9 deg; joints [-10.57, -45.058, 109.459, 136.487, 70.84, 107.307, -2381.899]
  MoveL 1139 to (-65.27, 210.27, 230) mm, rotated rx -180 ry 50 rz 127.3 deg; joints [-10.964, -45.141, 109.604, 136.104, 71.002, 107.392, -2377.303]
  MoveL 1140 to (-68.98, 216.33, 220) mm, rotated rx 180 ry 50 rz 122.34 deg; joints [-11.359, -45.225, 109.743, 135.719, 71.16, 107.481, -2372.338]
  MoveL 1141 to (-72.31, 223.11, 210) mm, rotated rx 180 ry 50 rz 117.03 deg; joints [-11.755, -45.309, 109.876, 135.332, 71.314, 107.573, -2367.029]
  MoveL 1142 to (-75.1, 230.56, 200) mm, rotated rx 180 ry 50 rz 111.4 deg; joints [-12.152, -45.394, 110.003, 134.943, 71.465, 107.668, -2361.404]
  MoveL 1143 to (-77.2, 238.6, 190) mm, rotated rx -180 ry 50 rz 105.49 deg; joints [-12.549, -45.477, 110.125, 134.553, 71.612, 107.766, -2355.49]
  MoveL 1144 to (-78.47, 247.13, 180) mm, rotated rx -180 ry 50 rz 99.32 deg; joints [-12.947, -45.561, 110.24, 134.161, 71.757, 107.867, -2349.316]
  MoveL 1145 to (-78.79, 256, 170) mm, rotated rx -180 ry 50 rz 92.91 deg; joints [-13.346, -45.643, 110.35, 133.768, 71.898, 107.971, -2342.909]
  MoveL 1146 to (-78.09, 265.05, 160) mm, rotated rx 180 ry 50 rz 86.3 deg; joints [-13.746, -45.723, 110.453, 133.374, 72.038, 108.077, -2336.299]
  MoveL 1147 to (-76.31, 274.12, 150) mm, rotated rx 180 ry 50 rz 79.52 deg; joints [-14.146, -45.801, 110.55, 132.979, 72.175, 108.186, -2329.517]
  MoveL 1148 to (-73.44, 283.02, 140) mm, rotated rx 180 ry 50 rz 72.6 deg; joints [-14.546, -45.876, 110.641, 132.583, 72.311, 108.295, -2322.596]
  MoveL 1149 to (-69.5, 291.57, 130) mm, rotated rx 180 ry 50 rz 65.57 deg; joints [-14.948, -45.947, 110.725, 132.187, 72.447, 108.406, -2315.57]
  MoveL 1150 to (-64.57, 299.61, 120) mm, rotated rx 180 ry 50 rz 58.48 deg; joints [-15.349, -46.014, 110.803, 131.79, 72.582, 108.517, -2308.477]
  MoveL 1151 to (-58.74, 306.97, 110) mm, rotated rx 180 ry 50 rz 51.35 deg; joints [-15.751, -46.075, 110.874, 131.393, 72.717, 108.628, -2301.355]
  MoveL 1152 to (-52.14, 313.53, 100) mm, rotated rx 180 ry 50 rz 44.25 deg; joints [-16.154, -46.13, 110.939, 130.996, 72.852, 108.738, -2294.246]
  MoveL 1153 to (-44.91, 319.19, 90) mm, rotated rx 180 ry 50 rz 37.19 deg; joints [-16.557, -46.179, 110.998, 130.599, 72.988, 108.848, -2287.194]
  MoveL 1154 to (-37.24, 323.88, 80) mm, rotated rx 180 ry 50 rz 30.24 deg; joints [-16.96, -46.221, 111.05, 130.202, 73.125, 108.957, -2280.242]
  MoveL 1155 to (-29.3, 327.59, 70) mm, rotated rx -180 ry 50 rz 23.44 deg; joints [-17.364, -46.256, 111.095, 129.806, 73.263, 109.064, -2273.438]
  MoveL 1156 to (-21.27, 330.31, 60) mm, rotated rx 180 ry 50 rz 16.83 deg; joints [-17.768, -46.285, 111.133, 129.41, 73.401, 109.17, -2266.828]
  MoveL 1157 to (-13.31, 332.11, 50) mm, rotated rx -180 ry 50 rz 10.46 deg; joints [-18.172, -46.306, 111.165, 129.014, 73.541, 109.275, -2260.456]
  MoveL 1158 to (-5.58, 333.04, 40) mm, rotated rx -180 ry 50 rz 4.37 deg; joints [-18.576, -46.322, 111.19, 128.619, 73.681, 109.379, -2254.37]
  MoveL 1159 to (1.77, 333.22, 30) mm, rotated rx 180 ry 50 rz -1.39 deg; joints [-18.981, -46.331, 111.209, 128.224, 73.821, 109.482, -2248.612]
  MoveL 1160 to (8.64, 332.76, 20) mm, rotated rx 180 ry 50 rz -6.77 deg; joints [-19.385, -46.334, 111.222, 127.829, 73.962, 109.585, -2243.227]
  MoveL 1161 to (14.93, 331.81, 10) mm, rotated rx 180 ry 50 rz -11.75 deg; joints [-19.79, -46.333, 111.228, 127.434, 74.102, 109.689, -2238.254]
  MoveL 1162 to (20.57, 330.51, 0) mm, rotated rx 180 ry 50 rz -16.27 deg; joints [-20.194, -46.328, 111.227, 127.04, 74.242, 109.792, -2233.733]
  MoveL 1163 to (-43.85, 188.95, 290) mm, rotated rx -180 ry 50 rz 148.32 deg; joints [-8.613, -44.637, 108.645, 138.378, 69.974, 106.924, -2398.321]
  Set speed (60.0 mm/s)
  MoveL 1164 to (-28.22, 202.67, 290) mm, rotated rx -180 ry 50 rz 153.79 deg; joints [-8.613, -45.711, 108.751, 138.138, 69.253, 107.611, -2403.793]
  MoveL 1165 to (20.57, 330.51, 0) mm, rotated rx -180 ry 50 rz -16.27 deg; joints [-20.194, -46.328, 111.227, 127.04, 74.242, 109.792, -2233.733]
  Set speed (60.0 mm/s)
  MoveL 1166 to (10.16, 312.5, 0) mm, rotated rx 180 ry 50 rz -10.95 deg; joints [-20.194, -47.443, 111.32, 126.804, 73.628, 110.643, -2239.047]
  MoveL 1167 to (20.57, 330.51, 0) mm, rotated rx 180 ry 50 rz -16.27 deg; joints [-20.194, -46.328, 111.227, 127.04, 74.242, 109.792, -2233.733]
  Set speed (60.0 mm/s)
  MoveL 1168 to (14.93, 331.81, 10) mm, rotated rx -180 ry 50 rz -11.75 deg; joints [-19.79, -46.333, 111.228, 127.434, 74.102, 109.689, -2238.254]
  MoveL 1169 to (8.64, 332.76, 20) mm, rotated rx -180 ry 50 rz -6.77 deg; joints [-19.385, -46.334, 111.222, 127.829, 73.962, 109.585, -2243.227]
  MoveL 1170 to (1.77, 333.22, 30) mm, rotated rx 180 ry 50 rz -1.39 deg; joints [-18.981, -46.331, 111.209, 128.224, 73.821, 109.482, -2248.612]
  MoveL 1171 to (-5.58, 333.04, 40) mm, rotated rx 180 ry 50 rz 4.37 deg; joints [-18.576, -46.322, 111.19, 128.619, 73.681, 109.379, -2254.37]
  MoveL 1172 to (-13.31, 332.11, 50) mm, rotated rx -180 ry 50 rz 10.46 deg; joints [-18.172, -46.306, 111.165, 129.014, 73.541, 109.275, -2260.456]
  MoveL 1173 to (-21.27, 330.31, 60) mm, rotated rx 180 ry 50 rz 16.83 deg; joints [-17.768, -46.285, 111.133, 129.41, 73.401, 109.17, -2266.828]
  MoveL 1174 to (-29.3, 327.59, 70) mm, rotated rx 180 ry 50 rz 23.44 deg; joints [-17.364, -46.256, 111.095, 129.806, 73.263, 109.064, -2273.438]
  MoveL 1175 to (-37.24, 323.88, 80) mm, rotated rx -180 ry 50 rz 30.24 deg; joints [-16.96, -46.221, 111.05, 130.202, 73.125, 108.957, -2280.242]
  MoveL 1176 to (-44.91, 319.19, 90) mm, rotated rx 180 ry 50 rz 37.19 deg; joints [-16.557, -46.179, 110.998, 130.599, 72.988, 108.848, -2287.194]
  MoveL 1177 to (-52.14, 313.53, 100) mm, rotated rx -180 ry 50 rz 44.25 deg; joints [-16.154, -46.13, 110.939, 130.996, 72.852, 108.738, -2294.246]
  MoveL 1178 to (-58.74, 306.97, 110) mm, rotated rx 180 ry 50 rz 51.35 deg; joints [-15.751, -46.075, 110.874, 131.393, 72.717, 108.628, -2301.355]
  MoveL 1179 to (-64.57, 299.61, 120) mm, rotated rx 180 ry 50 rz 58.48 deg; joints [-15.349, -46.014, 110.803, 131.79, 72.582, 108.517, -2308.477]
  MoveL 1180 to (-69.5, 291.57, 130) mm, rotated rx 180 ry 50 rz 65.57 deg; joints [-14.948, -45.947, 110.725, 132.187, 72.447, 108.406, -2315.57]
  MoveL 1181 to (-73.44, 283.02, 140) mm, rotated rx 180 ry 50 rz 72.6 deg; joints [-14.546, -45.876, 110.641, 132.583, 72.311, 108.295, -2322.596]
  MoveL 1182 to (-76.31, 274.12, 150) mm, rotated rx -180 ry 50 rz 79.52 deg; joints [-14.146, -45.801, 110.55, 132.979, 72.175, 108.186, -2329.517]
  MoveL 1183 to (-78.09, 265.05, 160) mm, rotated rx 180 ry 50 rz 86.3 deg; joints [-13.746, -45.723, 110.453, 133.374, 72.038, 108.077, -2336.299]
  MoveL 1184 to (-78.79, 256, 170) mm, rotated rx 180 ry 50 rz 92.91 deg; joints [-13.346, -45.643, 110.35, 133.768, 71.898, 107.971, -2342.909]
  MoveL 1185 to (-78.47, 247.13, 180) mm, rotated rx -180 ry 50 rz 99.32 deg; joints [-12.947, -45.561, 110.24, 134.161, 71.757, 107.867, -2349.316]
  MoveL 1186 to (-77.2, 238.6, 190) mm, rotated rx 180 ry 50 rz 105.49 deg; joints [-12.549, -45.477, 110.125, 134.553, 71.612, 107.766, -2355.49]
  MoveL 1187 to (-75.1, 230.56, 200) mm, rotated rx -180 ry 50 rz 111.4 deg; joints [-12.152, -45.394, 110.003, 134.943, 71.465, 107.668, -2361.404]
  MoveL 1188 to (-72.31, 223.11, 210) mm, rotated rx 180 ry 50 rz 117.03 deg; joints [-11.755, -45.309, 109.876, 135.332, 71.314, 107.573, -2367.029]
  MoveL 1189 to (-68.98, 216.33, 220) mm, rotated rx 180 ry 50 rz 122.34 deg; joints [-11.359, -45.225, 109.743, 135.719, 71.16, 107.481, -2372.338]
  MoveL 1190 to (-65.27, 210.27, 230) mm, rotated rx 180 ry 50 rz 127.3 deg; joints [-10.964, -45.141, 109.604, 136.104, 71.002, 107.392, -2377.303]
  MoveL 1191 to (-61.34, 204.96, 240) mm, rotated rx -180 ry 50 rz 131.9 deg; joints [-10.57, -45.058, 109.459, 136.487, 70.84, 107.307, -2381.899]
  MoveL 1192 to (-57.36, 200.4, 250) mm, rotated rx -180 ry 50 rz 136.1 deg; joints [-10.177, -44.974, 109.308, 136.869, 70.674, 107.224, -2386.095]
  MoveL 1193 to (-53.49, 196.56, 260) mm, rotated rx 180 ry 50 rz 139.86 deg; joints [-9.784, -44.89, 109.151, 137.249, 70.505, 107.145, -2389.865]
  MoveL 1194 to (-49.86, 193.4, 270) mm, rotated rx 180 ry 50 rz 143.18 deg; joints [-9.393, -44.806, 108.988, 137.627, 70.332, 107.069, -2393.179]
  MoveL 1195 to (-46.6, 190.89, 280) mm, rotated rx 180 ry 50 rz 146.01 deg; joints [-9.003, -44.722, 108.819, 138.003, 70.155, 106.995, -2396.008]
  MoveL 1196 to (-43.85, 188.95, 290) mm, rotated rx -180 ry 50 rz 148.32 deg; joints [-8.613, -44.637, 108.645, 138.378, 69.974, 106.924, -2398.321]
  MoveL 1197 to (-28.22, 202.67, 290) mm, rotated rx -180 ry 50 rz 153.79 deg; joints [-8.613, -45.711, 108.751, 138.138, 69.253, 107.611, -2403.793]
  Set speed (60.0 mm/s)
  MoveL 1198 to (-30.4, 203.93, 280) mm, rotated rx -180 ry 50 rz 151.53 deg; joints [-9.003, -45.797, 108.926, 137.764, 69.437, 107.687, -2401.533]
  MoveL 1199 to (-33, 205.58, 270) mm, rotated rx -180 ry 50 rz 148.77 deg; joints [-9.393, -45.881, 109.094, 137.388, 69.617, 107.765, -2398.768]
  MoveL 1200 to (-35.92, 207.69, 260) mm, rotated rx 180 ry 50 rz 145.53 deg; joints [-9.784, -45.965, 109.256, 137.011, 69.795, 107.846, -2395.528]
  MoveL 1201 to (-39.07, 210.28, 250) mm, rotated rx 180 ry 50 rz 141.84 deg; joints [-10.177, -46.049, 109.413, 136.631, 69.968, 107.93, -2391.841]
  MoveL 1202 to (-42.34, 213.41, 240) mm, rotated rx 180 ry 50 rz 137.73 deg; joints [-10.57, -46.132, 109.563, 136.25, 70.138, 108.017, -2387.735]
  MoveL 1203 to (-45.62, 217.1, 230) mm, rotated rx -180 ry 50 rz 133.24 deg; joints [-10.964, -46.215, 109.708, 135.867, 70.304, 108.106, -2383.236]
  MoveL 1204 to (-48.8, 221.36, 220) mm, rotated rx 180 ry 50 rz 128.37 deg; joints [-11.359, -46.299, 109.846, 135.482, 70.467, 108.199, -2378.371]
  MoveL 1205 to (-51.74, 226.19, 210) mm, rotated rx 180 ry 50 rz 123.16 deg; joints [-11.755, -46.382, 109.978, 135.096, 70.625, 108.296, -2373.164]
  MoveL 1206 to (-54.33, 231.55, 200) mm, rotated rx 180 ry 50 rz 117.64 deg; joints [-12.152, -46.466, 110.105, 134.707, 70.781, 108.395, -2367.64]
  MoveL 1207 to (-56.44, 237.4, 190) mm, rotated rx 180 ry 50 rz 111.82 deg; joints [-12.549, -46.549, 110.225, 134.318, 70.932, 108.498, -2361.825]
  MoveL 1208 to (-57.96, 243.66, 180) mm, rotated rx -180 ry 50 rz 105.74 deg; joints [-12.947, -46.632, 110.34, 133.926, 71.081, 108.604, -2355.742]
  MoveL 1209 to (-58.8, 250.25, 170) mm, rotated rx -180 ry 50 rz 99.42 deg; joints [-13.346, -46.715, 110.448, 133.533, 71.226, 108.713, -2349.418]
  MoveL 1210 to (-58.89, 257.04, 160) mm, rotated rx 180 ry 50 rz 92.88 deg; joints [-13.746, -46.795, 110.55, 133.139, 71.37, 108.825, -2342.877]
  MoveL 1211 to (-58.18, 263.92, 150) mm, rotated rx -180 ry 50 rz 86.15 deg; joints [-14.146, -46.874, 110.646, 132.744, 71.511, 108.939, -2336.149]
  MoveL 1212 to (-56.65, 270.74, 140) mm, rotated rx 180 ry 50 rz 79.26 deg; joints [-14.546, -46.951, 110.736, 132.348, 71.65, 109.055, -2329.263]
  MoveL 1213 to (-54.3, 277.38, 130) mm, rotated rx -180 ry 50 rz 72.25 deg; joints [-14.948, -47.023, 110.82, 131.951, 71.789, 109.171, -2322.251]
  MoveL 1214 to (-51.17, 283.7, 120) mm, rotated rx 180 ry 50 rz 65.15 deg; joints [-15.349, -47.092, 110.897, 131.554, 71.927, 109.289, -2315.149]
  MoveL 1215 to (-47.33, 289.58, 110) mm, rotated rx 180 ry 50 rz 57.99 deg; joints [-15.751, -47.156, 110.968, 131.157, 72.065, 109.407, -2307.994]
  MoveL 1216 to (-42.85, 294.92, 100) mm, rotated rx 180 ry 50 rz 50.83 deg; joints [-16.154, -47.214, 111.032, 130.76, 72.203, 109.524, -2300.828]
  MoveL 1217 to (-37.86, 299.62, 90) mm, rotated rx 180 ry 50 rz 43.7 deg; joints [-16.557, -47.266, 111.09, 130.363, 72.342, 109.641, -2293.695]
  MoveL 1218 to (-32.46, 303.64, 80) mm, rotated rx -180 ry 50 rz 36.64 deg; joints [-16.96, -47.312, 111.141, 129.966, 72.482, 109.757, -2286.643]
  MoveL 1219 to (-26.8, 306.94, 70) mm, rotated rx -180 ry 50 rz 29.72 deg; joints [-17.364, -47.351, 111.186, 129.569, 72.622, 109.871, -2279.72]
  MoveL 1220 to (-21, 309.52, 60) mm, rotated rx 180 ry 50 rz 22.98 deg; joints [-17.768, -47.383, 111.225, 129.173, 72.764, 109.984, -2272.977]
  MoveL 1221 to (-15.19, 311.39, 50) mm, rotated rx 180 ry 50 rz 16.46 deg; joints [-18.172, -47.408, 111.257, 128.777, 72.907, 110.096, -2266.464]
  MoveL 1222 to (-9.5, 312.61, 40) mm, rotated rx 180 ry 50 rz 10.23 deg; joints [-18.576, -47.426, 111.282, 128.382, 73.05, 110.207, -2260.231]
  MoveL 1223 to (-4.03, 313.25, 30) mm, rotated rx 180 ry 50 rz 4.33 deg; joints [-18.981, -47.439, 111.301, 127.987, 73.194, 110.316, -2254.327]
  MoveL 1224 to (1.12, 313.37, 20) mm, rotated rx -180 ry 50 rz -1.2 deg; joints [-19.385, -47.445, 111.314, 127.593, 73.339, 110.425, -2248.799]
  MoveL 1225 to (5.87, 313.09, 10) mm, rotated rx 180 ry 50 rz -6.31 deg; joints [-19.79, -47.446, 111.32, 127.198, 73.484, 110.534, -2243.692]
  MoveL 1226 to (10.16, 312.5, 0) mm, rotated rx 180 ry 50 rz -10.95 deg; joints [-20.194, -47.443, 111.32, 126.804, 73.628, 110.643, -2239.047]
  Set speed (1000.0 mm/s)
  MoveL 1227 to (10.16, 312.5, 0) mm, rotated rx 180 ry 50 rz -10.95 deg; joints [-20.194, -47.443, 111.32, 126.804, 73.628, 110.643, -2239.047]
